LIN {X 0,Y 178.963,Z 581.271,A -85,B 0,C 180,E1 -22404.933,E2 -22404.933} C_VEL
LIN {X 0,Y 179.094,Z 587.177,A -85,B 0,C 180,E1 -22407.754,E2 -22407.754} C_VEL
LIN {X 0,Y 179.064,Z 591.005,A -85,B 0,C 180,E1 -22410.003,E2 -22410.003} C_VEL
LIN {X 0,Y 178.631,Z 594.089,A -85,B 0,C 180,E1 -22412.257,E2 -22412.257} C_VEL
LIN {X 0,Y 177.778,Z 597.609,A -85,B 0,C 180,E1 -22415.674,E2 -22415.674} C_VEL
LIN {X 0,Y 177.413,Z 600.176,A -85,B 0,C 180,E1 -22419.12,E2 -22419.12} C_VEL
LIN {X 0,Y 177.958,Z 602.371,A -85,B 0,C 180,E1 -22423.709,E2 -22423.709} C_VEL
LIN {X 0,Y 180.059,Z 603.293,A -85,B 0,C 180,E1 -22428.198,E2 -22428.198} C_VEL
LIN {X 0,Y 183.553,Z 602.927,A -85,B 0,C 180,E1 -22432.515,E2 -22432.515} C_VEL
LIN {X 0,Y 188.306,Z 601.288,A -85,B 0,C 180,E1 -22436.609,E2 -22436.609} C_VEL
LIN {X 0,Y 194.454,Z 598.389,A -85,B 0,C 180,E1 -22440.4,E2 -22440.4} C_VEL
LIN {X 0,Y 201.914,Z 594.146,A -85,B 0,C 180,E1 -22443.845,E2 -22443.845} C_VEL
LIN {X 0,Y 210.351,Z 588.495,A -85,B 0,C 180,E1 -22446.972,E2 -22446.972} C_VEL
LIN {X 0,Y 217.836,Z 582.763,A -85,B 0,C 180,E1 -22449.257,E2 -22449.257} C_VEL
LIN {X 0,Y 227.369,Z 574.527,A -85,B 0,C 180,E1 -22451.651,E2 -22451.651} C_VEL
LIN {X 0,Y 235.426,Z 566.669,A -85,B 0,C 180,E1 -22453.364,E2 -22453.364} C_VEL
LIN {X 0,Y 244.098,Z 557.229,A -85,B 0,C 180,E1 -22454.864,E2 -22454.864} C_VEL
LIN {X 0,Y 253.168,Z 545.908,A -85,B 0,C 180,E1 -22456.203,E2 -22456.203} C_VEL
LIN {X 0,Y 251.587,Z 547.776,A -85,B 0,C 180,E1 -22456.707,E2 -22456.707} C_VEL
LIN {X 0,Y 243.286,Z 557.033,A -85,B 0,C 180,E1 -22458.362,E2 -22458.362} C_VEL
LIN {X 0,Y 235.512,Z 564.518,A -85,B 0,C 180,E1 -22460.089,E2 -22460.089} C_VEL
LIN {X 0,Y 228.038,Z 570.729,A -85,B 0,C 180,E1 -22461.947,E2 -22461.947} C_VEL
LIN {X 0,Y 220.975,Z 575.798,A -85,B 0,C 180,E1 -22463.957,E2 -22463.957} C_VEL
LIN {X 0,Y 212.204,Z 580.994,A -85,B 0,C 180,E1 -22466.875,E2 -22466.875} C_VEL
LIN {X 0,Y 206.132,Z 583.851,A -85,B 0,C 180,E1 -22469.241,E2 -22469.241} C_VEL
LIN {X 0,Y 198.857,Z 586.335,A -85,B 0,C 180,E1 -22472.648,E2 -22472.648} C_VEL
LIN {X 0,Y 192.485,Z 587.392,A -85,B 0,C 180,E1 -22476.319,E2 -22476.319} C_VEL
LIN {X 0,Y 187.209,Z 586.992,A -85,B 0,C 180,E1 -22480.253,E2 -22480.253} C_VEL
LIN {X 0,Y 182.885,Z 585.199,A -85,B 0,C 180,E1 -22484.395,E2 -22484.395} C_VEL
LIN {X 0,Y 181.145,Z 583.766,A -85,B 0,C 180,E1 -22486.539,E2 -22486.539} C_VEL
LIN {X 0,Y 178.883,Z 579.753,A -85,B 0,C 180,E1 -22490.958,E2 -22490.958} C_VEL
LIN {X 0,Y 177.692,Z 575.71,A -85,B 0,C 180,E1 -22494.325,E2 -22494.325} C_VEL
LIN {X 0,Y 176.868,Z 568.695,A -85,B 0,C 180,E1 -22498.861,E2 -22498.861} C_VEL
LIN {X 0,Y 176.997,Z 560.839,A -85,B 0,C 180,E1 -22502.845,E2 -22502.845} C_VEL
LIN {X 0,Y 177.27,Z 552.453,A -85,B 0,C 180,E1 -22506.249,E2 -22506.249} C_VEL
LIN {X 0,Y 177.78,Z 543.801,A -85,B 0,C 180,E1 -22509.158,E2 -22509.158} C_VEL
LIN {X 0,Y 178.492,Z 533.877,A -85,B 0,C 180,E1 -22511.93,E2 -22511.93} C_VEL
LIN {X 0,Y 179.517,Z 521.445,A -85,B 0,C 180,E1 -22514.742,E2 -22514.742} C_VEL
LIN {X 0,Y 180.559,Z 509.146,A -85,B 0,C 180,E1 -22516.973,E2 -22516.973} C_VEL
LIN {X 0,Y 181.504,Z 495.349,A -85,B 0,C 180,E1 -22518.922,E2 -22518.922} C_VEL
LIN {X 0,Y 182.391,Z 480.871,A -85,B 0,C 180,E1 -22520.438,E2 -22520.438} C_VEL
LIN {X 0,Y 184.893,Z 424.724,A -85,B 0,C 180,E1 -22524.498,E2 -22524.498} C_VEL
LIN {X 0,Y 185.569,Z 410.627,A -85,B 0,C 180,E1 -22525.472,E2 -22525.472} C_VEL
LIN {X 0,Y 178.743,Z 384.831,A -85,B 0,C 180,E1 -22527.528,E2 -22527.528} C_VEL
LIN {X 0,Y 178.643,Z 384.231,A -85,B 0,C 180,E1 -22527.61,E2 -22527.61} C_VEL
LIN {X 0,Y 178.494,Z 384.245,A -85,B 0,C 180,E1 -22533.452,E2 -22533.452} C_VEL
LIN {X 0,Y 178.401,Z 384.26,A -85,B 0,C 180,E1 -22539.073,E2 -22539.073} C_VEL
LIN {X 0,Y 178.404,Z 384.258,A -85,B 0,C 180,E1 -22542.043,E2 -22542.043} C_VEL
LIN {X 0,Y 178.399,Z 384.261,A -85,B 0,C 180,E1 -22545.162,E2 -22545.162} C_VEL
LIN {X 0,Y 178.415,Z 384.259,A -85,B 0,C 180,E1 -22548.455,E2 -22548.455} C_VEL
LIN {X 0,Y 178.468,Z 384.251,A -85,B 0,C 180,E1 -22551.961,E2 -22551.961} C_VEL
LIN {X 0,Y 178.495,Z 384.249,A -85,B 0,C 180,E1 -22556.546,E2 -22556.546} C_VEL
LIN {X 0,Y 178.527,Z 384.242,A -85,B 0,C 180,E1 -22560.004,E2 -22560.004} C_VEL
LIN {X 0,Y 178.538,Z 384.244,A -85,B 0,C 180,E1 -22564.873,E2 -22564.873} C_VEL
LIN {X 0,Y 178.627,Z 384.233,A -85,B 0,C 180,E1 -22570.781,E2 -22570.781} C_VEL
LIN {X 0,Y 178.662,Z 384.225,A -85,B 0,C 180,E1 -22576.346,E2 -22576.346} C_VEL
LIN {X 0,Y 178.914,Z 384.197,A -85,B 0,C 180,E1 -22580.957,E2 -22580.957} C_VEL
LIN {X 0,Y 179.155,Z 384.166,A -85,B 0,C 180,E1 -22587.749,E2 -22587.749} C_VEL
LIN {X 0,Y 179.374,Z 384.143,A -85,B 0,C 180,E1 -22589.997,E2 -22589.997} C_VEL
LIN {X 0,Y 178.878,Z 384.198,A -85,B 0,C 180,E1 -22594.504,E2 -22594.504} C_VEL
LIN {X 0,Y 178.978,Z 384.189,A -85,B 0,C 180,E1 -22599.034,E2 -22599.034} C_VEL
LIN {X 0,Y 178.686,Z 384.222,A -85,B 0,C 180,E1 -22603.647,E2 -22603.647} C_VEL
LIN {X 0,Y 178.648,Z 384.231,A -85,B 0,C 180,E1 -22608.341,E2 -22608.341} C_VEL
LIN {X 0,Y 178.509,Z 384.245,A -85,B 0,C 180,E1 -22613.182,E2 -22613.182} C_VEL
LIN {X 0,Y 178.484,Z 384.25,A -85,B 0,C 180,E1 -22618.194,E2 -22618.194} C_VEL
LIN {X 0,Y 178.475,Z 384.246,A -85,B 0,C 180,E1 -22620.788,E2 -22620.788} C_VEL
LIN {X 0,Y 178.481,Z 384.252,A -85,B 0,C 180,E1 -22624.217,E2 -22624.217} C_VEL
LIN {X 0,Y 178.48,Z 384.248,A -85,B 0,C 180,E1 -22629.049,E2 -22629.049} C_VEL
LIN {X 0,Y 178.509,Z 384.249,A -85,B 0,C 180,E1 -22632.009,E2 -22632.009} C_VEL
LIN {X 0,Y 178.524,Z 384.246,A -85,B 0,C 180,E1 -22635.118,E2 -22635.118} C_VEL
LIN {X 0,Y 178.513,Z 384.243,A -85,B 0,C 180,E1 -22638.415,E2 -22638.415} C_VEL
LIN {X 0,Y 178.481,Z 384.253,A -85,B 0,C 180,E1 -22643.797,E2 -22643.797} C_VEL
LIN {X 0,Y 178.484,Z 384.246,A -85,B 0,C 180,E1 -22646.546,E2 -22646.546} C_VEL
LIN {X 0,Y 178.515,Z 384.248,A -85,B 0,C 180,E1 -22650.005,E2 -22650.005} C_VEL
LIN {X 0,Y 178.527,Z 384.243,A -85,B 0,C 180,E1 -22654.875,E2 -22654.875} C_VEL
LIN {X 0,Y 178.615,Z 384.235,A -85,B 0,C 180,E1 -22660.783,E2 -22660.783} C_VEL
LIN {X 0,Y 178.673,Z 384.226,A -85,B 0,C 180,E1 -22666.349,E2 -22666.349} C_VEL
LIN {X 0,Y 178.97,Z 384.19,A -85,B 0,C 180,E1 -22670.963,E2 -22670.963} C_VEL
LIN {X 0,Y 179.148,Z 384.17,A -85,B 0,C 180,E1 -22677.752,E2 -22677.752} C_VEL
LIN {X 0,Y 179.364,Z 384.14,A -85,B 0,C 180,E1 -22680,E2 -22680} C_VEL
LIN {X 0,Y 178.87,Z 384.201,A -85,B 0,C 180,E1 -22684.507,E2 -22684.507} C_VEL
LIN {X 0,Y 178.97,Z 384.19,A -85,B 0,C 180,E1 -22689.038,E2 -22689.038} C_VEL
LIN {X 0,Y 178.68,Z 384.228,A -85,B 0,C 180,E1 -22693.651,E2 -22693.651} C_VEL
LIN {X 0,Y 178.663,Z 384.226,A -85,B 0,C 180,E1 -22698.343,E2 -22698.343} C_VEL
LIN {X 0,Y 178.506,Z 384.249,A -85,B 0,C 180,E1 -22703.186,E2 -22703.186} C_VEL
LIN {X 0,Y 178.478,Z 384.246,A -85,B 0,C 180,E1 -22708.199,E2 -22708.199} C_VEL
LIN {X 0,Y 178.47,Z 384.251,A -85,B 0,C 180,E1 -22710.793,E2 -22710.793} C_VEL
LIN {X 0,Y 178.478,Z 384.251,A -85,B 0,C 180,E1 -22714.221,E2 -22714.221} C_VEL
LIN {X 0,Y 178.49,Z 384.249,A -85,B 0,C 180,E1 -22719.05,E2 -22719.05} C_VEL
LIN {X 0,Y 178.515,Z 384.247,A -85,B 0,C 180,E1 -22722.012,E2 -22722.012} C_VEL
LIN {X 0,Y 178.525,Z 384.244,A -85,B 0,C 180,E1 -22725.122,E2 -22725.122} C_VEL
LIN {X 0,Y 178.512,Z 384.246,A -85,B 0,C 180,E1 -22728.42,E2 -22728.42} C_VEL
LIN {X 0,Y 178.785,Z 384.32,A -85,B 0,C 180,E1 -22735.035,E2 -22735.035} C_VEL
LIN {X 0,Y 181.805,Z 398.712,A -85,B 0,C 180,E1 -22741.314,E2 -22741.314} C_VEL
LIN {X 0,Y 182.169,Z 424.055,A -85,B 0,C 180,E1 -22743.124,E2 -22743.124} C_VEL
LIN {X 0,Y 184.78,Z 459.469,A -85,B 0,C 180,E1 -22745.699,E2 -22745.699} C_VEL
LIN {X 0,Y 182.685,Z 509.123,A -85,B 0,C 180,E1 -22749.378,E2 -22749.378} C_VEL
LIN {X 0,Y 182.078,Z 520.419,A -85,B 0,C 180,E1 -22750.557,E2 -22750.557} C_VEL
LIN {X 0,Y 181.174,Z 532.641,A -85,B 0,C 180,E1 -22752.216,E2 -22752.216} C_VEL
LIN {X 0,Y 180.286,Z 545.376,A -85,B 0,C 180,E1 -22754.457,E2 -22754.457} C_VEL
LIN {X 0,Y 179.53,Z 556.851,A -85,B 0,C 180,E1 -22756.995,E2 -22756.995} C_VEL
LIN {X 0,Y 179.034,Z 567.273,A -85,B 0,C 180,E1 -22759.861,E2 -22759.861} C_VEL
LIN {X 0,Y 178.932,Z 573.096,A -85,B 0,C 180,E1 -22761.758,E2 -22761.758} C_VEL
LIN {X 0,Y 178.207,Z 576.828,A -85,B 0,C 180,E1 -22763.223,E2 -22763.223} C_VEL
LIN {X 0,Y 175.554,Z 582.018,A -85,B 0,C 180,E1 -22765.819,E2 -22765.819} C_VEL
LIN {X 0,Y 172.593,Z 587.441,A -85,B 0,C 180,E1 -22769.225,E2 -22769.225} C_VEL
LIN {X 0,Y 172.256,Z 589.213,A -85,B 0,C 180,E1 -22770.414,E2 -22770.414} C_VEL
LIN {X 0,Y 171.912,Z 591.86,A -85,B 0,C 180,E1 -22772.346,E2 -22772.346} C_VEL
LIN {X 0,Y 170.974,Z 595.636,A -85,B 0,C 180,E1 -22775.901,E2 -22775.901} C_VEL
LIN {X 0,Y 170.568,Z 598.473,A -85,B 0,C 180,E1 -22779.489,E2 -22779.489} C_VEL
LIN {X 0,Y 171.167,Z 600.987,A -85,B 0,C 180,E1 -22784.265,E2 -22784.265} C_VEL
LIN {X 0,Y 173.363,Z 602.236,A -85,B 0,C 180,E1 -22788.927,E2 -22788.927} C_VEL
LIN {X 0,Y 177.015,Z 602.255,A -85,B 0,C 180,E1 -22793.395,E2 -22793.395} C_VEL
LIN {X 0,Y 181.985,Z 601.049,A -85,B 0,C 180,E1 -22797.611,E2 -22797.611} C_VEL
LIN {X 0,Y 188.369,Z 598.627,A -85,B 0,C 180,E1 -22801.492,E2 -22801.492} C_VEL
LIN {X 0,Y 196.103,Z 594.92,A -85,B 0,C 180,E1 -22804.991,E2 -22804.991} C_VEL
LIN {X 0,Y 204.813,Z 589.857,A -85,B 0,C 180,E1 -22808.148,E2 -22808.148} C_VEL
LIN {X 0,Y 214.431,Z 583.262,A -85,B 0,C 180,E1 -22810.96,E2 -22810.96} C_VEL
LIN {X 0,Y 223.605,Z 576.089,A -85,B 0,C 180,E1 -22813.129,E2 -22813.129} C_VEL
LIN {X 0,Y 231.913,Z 568.759,A -85,B 0,C 180,E1 -22814.798,E2 -22814.798} C_VEL
LIN {X 0,Y 241.255,Z 559.52,A -85,B 0,C 180,E1 -22816.309,E2 -22816.309} C_VEL
LIN {X 0,Y 242.337,Z 558.359,A -85,B 0,C 180,E1 -22816.473,E2 -22816.473} C_VEL
LIN {X 0,Y 241.229,Z 559.378,A -85,B 0,C 180,E1 -22816.85,E2 -22816.85} C_VEL
LIN {X 0,Y 231.935,Z 567.506,A -85,B 0,C 180,E1 -22818.771,E2 -22818.771} C_VEL
LIN {X 0,Y 222.926,Z 574.186,A -85,B 0,C 180,E1 -22820.911,E2 -22820.911} C_VEL
LIN {X 0,Y 213.281,Z 580.016,A -85,B 0,C 180,E1 -22823.62,E2 -22823.62} C_VEL
LIN {X 0,Y 204.438,Z 584.223,A -85,B 0,C 180,E1 -22826.63,E2 -22826.63} C_VEL
LIN {X 0,Y 196.376,Z 586.894,A -85,B 0,C 180,E1 -22829.931,E2 -22829.931} C_VEL
LIN {X 0,Y 189.254,Z 588.163,A -85,B 0,C 180,E1 -22833.537,E2 -22833.537} C_VEL
LIN {X 0,Y 183.156,Z 588.055,A -85,B 0,C 180,E1 -22837.436,E2 -22837.436} C_VEL
LIN {X 0,Y 178.15,Z 586.509,A -85,B 0,C 180,E1 -22841.603,E2 -22841.603} C_VEL
LIN {X 0,Y 174.259,Z 583.552,A -85,B 0,C 180,E1 -22845.996,E2 -22845.996} C_VEL
LIN {X 0,Y 171.903,Z 579.165,A -85,B 0,C 180,E1 -22850.588,E2 -22850.588} C_VEL
LIN {X 0,Y 170.703,Z 574.779,A -85,B 0,C 180,E1 -22854.092,E2 -22854.092} C_VEL
LIN {X 0,Y 169.924,Z 568.358,A -85,B 0,C 180,E1 -22858.222,E2 -22858.222} C_VEL
LIN {X 0,Y 169.983,Z 560.308,A -85,B 0,C 180,E1 -22862.369,E2 -22862.369} C_VEL
LIN {X 0,Y 170.252,Z 551.734,A -85,B 0,C 180,E1 -22865.923,E2 -22865.923} C_VEL
LIN {X 0,Y 170.847,Z 541.719,A -85,B 0,C 180,E1 -22869.302,E2 -22869.302} C_VEL
LIN {X 0,Y 171.676,Z 530.406,A -85,B 0,C 180,E1 -22872.411,E2 -22872.411} C_VEL
LIN {X 0,Y 172.687,Z 518.564,A -85,B 0,C 180,E1 -22875.037,E2 -22875.037} C_VEL
LIN {X 0,Y 173.737,Z 505.427,A -85,B 0,C 180,E1 -22877.357,E2 -22877.357} C_VEL
LIN {X 0,Y 174.736,Z 490.405,A -85,B 0,C 180,E1 -22879.379,E2 -22879.379} C_VEL
LIN {X 0,Y 175.616,Z 474.732,A -85,B 0,C 180,E1 -22880.88,E2 -22880.88} C_VEL
LIN {X 0,Y 178.467,Z 411.765,A -85,B 0,C 180,E1 -22885.566,E2 -22885.566} C_VEL
LIN {X 0,Y 171.642,Z 385.486,A -85,B 0,C 180,E1 -22887.731,E2 -22887.731} C_VEL
LIN {X 0,Y 171.599,Z 385.109,A -85,B 0,C 180,E1 -22887.786,E2 -22887.786} C_VEL
LIN {X 0,Y 171.424,Z 385.128,A -85,B 0,C 180,E1 -22892.206,E2 -22892.206} C_VEL
LIN {X 0,Y 171.399,Z 385.132,A -85,B 0,C 180,E1 -22895.033,E2 -22895.033} C_VEL
LIN {X 0,Y 171.363,Z 385.137,A -85,B 0,C 180,E1 -22898.806,E2 -22898.806} C_VEL
LIN {X 0,Y 171.326,Z 385.143,A -85,B 0,C 180,E1 -22904.215,E2 -22904.215} C_VEL
LIN {X 0,Y 171.349,Z 385.137,A -85,B 0,C 180,E1 -22908.982,E2 -22908.982} C_VEL
LIN {X 0,Y 171.418,Z 385.129,A -85,B 0,C 180,E1 -22912.046,E2 -22912.046} C_VEL
LIN {X 0,Y 171.415,Z 385.131,A -85,B 0,C 180,E1 -22915.084,E2 -22915.084} C_VEL
LIN {X 0,Y 171.454,Z 385.126,A -85,B 0,C 180,E1 -22920.532,E2 -22920.532} C_VEL
LIN {X 0,Y 171.462,Z 385.126,A -85,B 0,C 180,E1 -22925.799,E2 -22925.799} C_VEL
LIN {X 0,Y 171.583,Z 385.11,A -85,B 0,C 180,E1 -22930.869,E2 -22930.869} C_VEL
LIN {X 0,Y 171.58,Z 385.11,A -85,B 0,C 180,E1 -22935.77,E2 -22935.77} C_VEL
LIN {X 0,Y 171.85,Z 385.078,A -85,B 0,C 180,E1 -22940.582,E2 -22940.582} C_VEL
LIN {X 0,Y 171.819,Z 385.077,A -85,B 0,C 180,E1 -22945.305,E2 -22945.305} C_VEL
LIN {X 0,Y 172.336,Z 385.02,A -85,B 0,C 180,E1 -22949.997,E2 -22949.997} C_VEL
LIN {X 0,Y 171.827,Z 385.076,A -85,B 0,C 180,E1 -22954.689,E2 -22954.689} C_VEL
LIN {X 0,Y 171.91,Z 385.07,A -85,B 0,C 180,E1 -22959.409,E2 -22959.409} C_VEL
LIN {X 0,Y 171.609,Z 385.106,A -85,B 0,C 180,E1 -22964.222,E2 -22964.222} C_VEL
LIN {X 0,Y 171.543,Z 385.116,A -85,B 0,C 180,E1 -22969.56,E2 -22969.56} C_VEL
LIN {X 0,Y 171.466,Z 385.126,A -85,B 0,C 180,E1 -22975.614,E2 -22975.614} C_VEL
LIN {X 0,Y 171.438,Z 385.123,A -85,B 0,C 180,E1 -22980.584,E2 -22980.584} C_VEL
LIN {X 0,Y 171.435,Z 385.129,A -85,B 0,C 180,E1 -22985.021,E2 -22985.021} C_VEL
LIN {X 0,Y 171.433,Z 385.125,A -85,B 0,C 180,E1 -22988.839,E2 -22988.839} C_VEL
LIN {X 0,Y 171.447,Z 385.128,A -85,B 0,C 180,E1 -22994.172,E2 -22994.172} C_VEL
LIN {X 0,Y 171.429,Z 385.125,A -85,B 0,C 180,E1 -22999.009,E2 -22999.009} C_VEL
LIN {X 0,Y 171.437,Z 385.13,A -85,B 0,C 180,E1 -23002.054,E2 -23002.054} C_VEL
LIN {X 0,Y 171.434,Z 385.128,A -85,B 0,C 180,E1 -23005.07,E2 -23005.07} C_VEL
LIN {X 0,Y 171.442,Z 385.128,A -85,B 0,C 180,E1 -23010.533,E2 -23010.533} C_VEL
LIN {X 0,Y 171.45,Z 385.124,A -85,B 0,C 180,E1 -23015.801,E2 -23015.801} C_VEL
LIN {X 0,Y 171.571,Z 385.112,A -85,B 0,C 180,E1 -23020.871,E2 -23020.871} C_VEL
LIN {X 0,Y 171.586,Z 385.109,A -85,B 0,C 180,E1 -23025.774,E2 -23025.774} C_VEL
LIN {X 0,Y 171.902,Z 385.07,A -85,B 0,C 180,E1 -23030.588,E2 -23030.588} C_VEL
LIN {X 0,Y 171.82,Z 385.08,A -85,B 0,C 180,E1 -23035.308,E2 -23035.308} C_VEL
LIN {X 0,Y 172.327,Z 385.016,A -85,B 0,C 180,E1 -23040,E2 -23040} C_VEL
LIN {X 0,Y 171.82,Z 385.08,A -85,B 0,C 180,E1 -23044.693,E2 -23044.693} C_VEL
LIN {X 0,Y 171.902,Z 385.07,A -85,B 0,C 180,E1 -23049.412,E2 -23049.412} C_VEL
LIN {X 0,Y 171.605,Z 385.108,A -85,B 0,C 180,E1 -23054.225,E2 -23054.225} C_VEL
LIN {X 0,Y 171.55,Z 385.111,A -85,B 0,C 180,E1 -23059.576,E2 -23059.576} C_VEL
LIN {X 0,Y 171.461,Z 385.126,A -85,B 0,C 180,E1 -23065.618,E2 -23065.618} C_VEL
LIN {X 0,Y 171.433,Z 385.127,A -85,B 0,C 180,E1 -23070.587,E2 -23070.587} C_VEL
LIN {X 0,Y 171.402,Z 385.134,A -85,B 0,C 180,E1 -23075.033,E2 -23075.033} C_VEL
LIN {X 0,Y 171.441,Z 385.126,A -85,B 0,C 180,E1 -23078.847,E2 -23078.847} C_VEL
LIN {X 0,Y 171.45,Z 385.125,A -85,B 0,C 180,E1 -23084.176,E2 -23084.176} C_VEL
LIN {X 0,Y 171.433,Z 385.13,A -85,B 0,C 180,E1 -23089.014,E2 -23089.014} C_VEL
LIN {X 0,Y 171.759,Z 385.193,A -85,B 0,C 180,E1 -23095.141,E2 -23095.141} C_VEL
LIN {X 0,Y 174.463,Z 397.947,A -85,B 0,C 180,E1 -23101.01,E2 -23101.01} C_VEL
LIN {X 0,Y 174.826,Z 402.006,A -85,B 0,C 180,E1 -23101.324,E2 -23101.324} C_VEL
LIN {X 0,Y 174.995,Z 422.325,A -85,B 0,C 180,E1 -23102.846,E2 -23102.846} C_VEL
LIN {X 0,Y 177.645,Z 459.917,A -85,B 0,C 180,E1 -23105.708,E2 -23105.708} C_VEL
LIN {X 0,Y 175.628,Z 508.529,A -85,B 0,C 180,E1 -23109.507,E2 -23109.507} C_VEL
LIN {X 0,Y 175,Z 520.309,A -85,B 0,C 180,E1 -23110.806,E2 -23110.806} C_VEL
LIN {X 0,Y 174.046,Z 533.204,A -85,B 0,C 180,E1 -23112.677,E2 -23112.677} C_VEL
LIN {X 0,Y 173.248,Z 545.71,A -85,B 0,C 180,E1 -23115.015,E2 -23115.015} C_VEL
LIN {X 0,Y 172.539,Z 556.89,A -85,B 0,C 180,E1 -23117.656,E2 -23117.656} C_VEL
LIN {X 0,Y 172.158,Z 567.042,A -85,B 0,C 180,E1 -23120.605,E2 -23120.605} C_VEL
LIN {X 0,Y 172.027,Z 575.333,A -85,B 0,C 180,E1 -23123.552,E2 -23123.552} C_VEL
LIN {X 0,Y 172.268,Z 582.181,A -85,B 0,C 180,E1 -23126.494,E2 -23126.494} C_VEL
LIN {X 0,Y 172.329,Z 586.641,A -85,B 0,C 180,E1 -23128.834,E2 -23128.834} C_VEL
LIN {X 0,Y 172.256,Z 589.213,A -85,B 0,C 180,E1 -23130.414,E2 -23130.414} C_VEL
LIN {X 0,Y 171.81,Z 590.823,A -85,B 0,C 180,E1 -23131.598,E2 -23131.598} C_VEL
LIN {X 0,Y 170.804,Z 592.098,A -85,B 0,C 180,E1 -23132.793,E2 -23132.793} C_VEL
LIN {X 0,Y 167.929,Z 594.009,A -85,B 0,C 180,E1 -23135.219,E2 -23135.219} C_VEL
LIN {X 0,Y 165.072,Z 595.457,A -85,B 0,C 180,E1 -23137.782,E2 -23137.782} C_VEL
LIN {X 0,Y 163.869,Z 596.57,A -85,B 0,C 180,E1 -23139.805,E2 -23139.805} C_VEL
LIN {X 0,Y 163.779,Z 596.978,A -85,B 0,C 180,E1 -23140.492,E2 -23140.492} C_VEL
LIN {X 0,Y 164.423,Z 599.434,A -85,B 0,C 180,E1 -23144.863,E2 -23144.863} C_VEL
LIN {X 0,Y 166.719,Z 601.046,A -85,B 0,C 180,E1 -23149.712,E2 -23149.712} C_VEL
LIN {X 0,Y 170.527,Z 601.456,A -85,B 0,C 180,E1 -23154.342,E2 -23154.342} C_VEL
LIN {X 0,Y 175.747,Z 600.682,A -85,B 0,C 180,E1 -23158.68,E2 -23158.68} C_VEL
LIN {X 0,Y 182.364,Z 598.728,A -85,B 0,C 180,E1 -23162.655,E2 -23162.655} C_VEL
LIN {X 0,Y 190.362,Z 595.548,A -85,B 0,C 180,E1 -23166.21,E2 -23166.21} C_VEL
LIN {X 0,Y 199.335,Z 591.051,A -85,B 0,C 180,E1 -23169.395,E2 -23169.395} C_VEL
LIN {X 0,Y 209.219,Z 585.134,A -85,B 0,C 180,E1 -23172.211,E2 -23172.211} C_VEL
LIN {X 0,Y 218.617,Z 578.65,A -85,B 0,C 180,E1 -23174.366,E2 -23174.366} C_VEL
LIN {X 0,Y 227.078,Z 572.026,A -85,B 0,C 180,E1 -23176.022,E2 -23176.022} C_VEL
LIN {X 0,Y 231.547,Z 568.232,A -85,B 0,C 180,E1 -23176.76,E2 -23176.76} C_VEL
LIN {X 0,Y 223.107,Z 574.203,A -85,B 0,C 180,E1 -23178.584,E2 -23178.584} C_VEL
LIN {X 0,Y 215.287,Z 578.909,A -85,B 0,C 180,E1 -23180.463,E2 -23180.463} C_VEL
LIN {X 0,Y 207.915,Z 582.624,A -85,B 0,C 180,E1 -23182.523,E2 -23182.523} C_VEL
LIN {X 0,Y 198.755,Z 586.235,A -85,B 0,C 180,E1 -23185.544,E2 -23185.544} C_VEL
LIN {X 0,Y 190.391,Z 588.402,A -85,B 0,C 180,E1 -23188.883,E2 -23188.883} C_VEL
LIN {X 0,Y 182.994,Z 589.156,A -85,B 0,C 180,E1 -23192.557,E2 -23192.557} C_VEL
LIN {X 0,Y 176.649,Z 588.558,A -85,B 0,C 180,E1 -23196.556,E2 -23196.556} C_VEL
LIN {X 0,Y 171.44,Z 586.601,A -85,B 0,C 180,E1 -23200.855,E2 -23200.855} C_VEL
LIN {X 0,Y 167.391,Z 583.202,A -85,B 0,C 180,E1 -23205.409,E2 -23205.409} C_VEL
LIN {X 0,Y 164.947,Z 578.371,A -85,B 0,C 180,E1 -23210.187,E2 -23210.187} C_VEL
LIN {X 0,Y 163.716,Z 573.659,A -85,B 0,C 180,E1 -23213.839,E2 -23213.839} C_VEL
LIN {X 0,Y 162.966,Z 566.838,A -85,B 0,C 180,E1 -23218.146,E2 -23218.146} C_VEL
LIN {X 0,Y 163.065,Z 558.318,A -85,B 0,C 180,E1 -23222.47,E2 -23222.47} C_VEL
LIN {X 0,Y 163.369,Z 549.245,A -85,B 0,C 180,E1 -23226.174,E2 -23226.174} C_VEL
LIN {X 0,Y 163.982,Z 539.246,A -85,B 0,C 180,E1 -23229.511,E2 -23229.511} C_VEL
LIN {X 0,Y 164.804,Z 527.785,A -85,B 0,C 180,E1 -23232.624,E2 -23232.624} C_VEL
LIN {X 0,Y 165.853,Z 515.28,A -85,B 0,C 180,E1 -23235.357,E2 -23235.357} C_VEL
LIN {X 0,Y 166.792,Z 503.141,A -85,B 0,C 180,E1 -23237.471,E2 -23237.471} C_VEL
LIN {X 0,Y 167.681,Z 489.929,A -85,B 0,C 180,E1 -23239.272,E2 -23239.272} C_VEL
LIN {X 0,Y 168.527,Z 474.924,A -85,B 0,C 180,E1 -23240.761,E2 -23240.761} C_VEL
LIN {X 0,Y 171.372,Z 412.584,A -85,B 0,C 180,E1 -23245.662,E2 -23245.662} C_VEL
LIN {X 0,Y 164.916,Z 387.845,A -85,B 0,C 180,E1 -23247.768,E2 -23247.768} C_VEL
LIN {X 0,Y 164.536,Z 385.989,A -85,B 0,C 180,E1 -23247.975,E2 -23247.975} C_VEL
LIN {X 0,Y 164.333,Z 386.009,A -85,B 0,C 180,E1 -23253.777,E2 -23253.777} C_VEL
LIN {X 0,Y 164.3,Z 386.019,A -85,B 0,C 180,E1 -23256.788,E2 -23256.788} C_VEL
LIN {X 0,Y 164.296,Z 386.018,A -85,B 0,C 180,E1 -23259.914,E2 -23259.914} C_VEL
LIN {X 0,Y 164.285,Z 386.017,A -85,B 0,C 180,E1 -23263.34,E2 -23263.34} C_VEL
LIN {X 0,Y 164.297,Z 386.018,A -85,B 0,C 180,E1 -23266.807,E2 -23266.807} C_VEL
LIN {X 0,Y 164.31,Z 386.013,A -85,B 0,C 180,E1 -23270.346,E2 -23270.346} C_VEL
LIN {X 0,Y 164.348,Z 386.014,A -85,B 0,C 180,E1 -23274.34,E2 -23274.34} C_VEL
LIN {X 0,Y 164.395,Z 386,A -85,B 0,C 180,E1 -23279.133,E2 -23279.133} C_VEL
LIN {X 0,Y 164.42,Z 386.003,A -85,B 0,C 180,E1 -23284.692,E2 -23284.692} C_VEL
LIN {X 0,Y 164.488,Z 385.994,A -85,B 0,C 180,E1 -23290.048,E2 -23290.048} C_VEL
LIN {X 0,Y 164.527,Z 385.987,A -85,B 0,C 180,E1 -23295.147,E2 -23295.147} C_VEL
LIN {X 0,Y 164.771,Z 385.962,A -85,B 0,C 180,E1 -23300.174,E2 -23300.174} C_VEL
LIN {X 0,Y 164.834,Z 385.951,A -85,B 0,C 180,E1 -23302.648,E2 -23302.648} C_VEL
LIN {X 0,Y 165.05,Z 385.922,A -85,B 0,C 180,E1 -23307.557,E2 -23307.557} C_VEL
LIN {X 0,Y 165.299,Z 385.896,A -85,B 0,C 180,E1 -23309.997,E2 -23309.997} C_VEL
LIN {X 0,Y 164.778,Z 385.954,A -85,B 0,C 180,E1 -23314.891,E2 -23314.891} C_VEL
LIN {X 0,Y 164.863,Z 385.947,A -85,B 0,C 180,E1 -23317.345,E2 -23317.345} C_VEL
LIN {X 0,Y 164.779,Z 385.957,A -85,B 0,C 180,E1 -23321.195,E2 -23321.195} C_VEL
LIN {X 0,Y 164.504,Z 385.993,A -85,B 0,C 180,E1 -23327.398,E2 -23327.398} C_VEL
LIN {X 0,Y 164.471,Z 385.995,A -85,B 0,C 180,E1 -23329.986,E2 -23329.986} C_VEL
LIN {X 0,Y 164.39,Z 386.008,A -85,B 0,C 180,E1 -23336.131,E2 -23336.131} C_VEL
LIN {X 0,Y 164.372,Z 386.003,A -85,B 0,C 180,E1 -23341.226,E2 -23341.226} C_VEL
LIN {X 0,Y 164.357,Z 386.01,A -85,B 0,C 180,E1 -23346.769,E2 -23346.769} C_VEL
LIN {X 0,Y 164.37,Z 386.006,A -85,B 0,C 180,E1 -23349.889,E2 -23349.889} C_VEL
LIN {X 0,Y 164.385,Z 386.008,A -85,B 0,C 180,E1 -23353.381,E2 -23353.381} C_VEL
LIN {X 0,Y 164.391,Z 386.004,A -85,B 0,C 180,E1 -23356.841,E2 -23356.841} C_VEL
LIN {X 0,Y 164.371,Z 386.008,A -85,B 0,C 180,E1 -23360.315,E2 -23360.315} C_VEL
LIN {X 0,Y 164.363,Z 386.009,A -85,B 0,C 180,E1 -23364.328,E2 -23364.328} C_VEL
LIN {X 0,Y 164.384,Z 386.006,A -85,B 0,C 180,E1 -23369.133,E2 -23369.133} C_VEL
LIN {X 0,Y 164.409,Z 386.001,A -85,B 0,C 180,E1 -23374.693,E2 -23374.693} C_VEL
LIN {X 0,Y 164.477,Z 385.997,A -85,B 0,C 180,E1 -23380.05,E2 -23380.05} C_VEL
LIN {X 0,Y 164.528,Z 385.984,A -85,B 0,C 180,E1 -23385.15,E2 -23385.15} C_VEL
LIN {X 0,Y 164.844,Z 385.95,A -85,B 0,C 180,E1 -23390.181,E2 -23390.181} C_VEL
LIN {X 0,Y 164.77,Z 385.957,A -85,B 0,C 180,E1 -23395.107,E2 -23395.107} C_VEL
LIN {X 0,Y 165.289,Z 385.893,A -85,B 0,C 180,E1 -23400,E2 -23400} C_VEL
LIN {X 0,Y 164.77,Z 385.958,A -85,B 0,C 180,E1 -23404.894,E2 -23404.894} C_VEL
LIN {X 0,Y 164.845,Z 385.946,A -85,B 0,C 180,E1 -23409.819,E2 -23409.819} C_VEL
LIN {X 0,Y 164.551,Z 385.987,A -85,B 0,C 180,E1 -23414.849,E2 -23414.849} C_VEL
LIN {X 0,Y 164.468,Z 385.993,A -85,B 0,C 180,E1 -23419.99,E2 -23419.99} C_VEL
LIN {X 0,Y 164.386,Z 386.006,A -85,B 0,C 180,E1 -23426.135,E2 -23426.135} C_VEL
LIN {X 0,Y 164.367,Z 386.01,A -85,B 0,C 180,E1 -23431.229,E2 -23431.229} C_VEL
LIN {X 0,Y 164.347,Z 386.009,A -85,B 0,C 180,E1 -23436.776,E2 -23436.776} C_VEL
LIN {X 0,Y 164.374,Z 386.008,A -85,B 0,C 180,E1 -23439.893,E2 -23439.893} C_VEL
LIN {X 0,Y 164.389,Z 386.007,A -85,B 0,C 180,E1 -23443.387,E2 -23443.387} C_VEL
LIN {X 0,Y 164.391,Z 386.002,A -85,B 0,C 180,E1 -23446.845,E2 -23446.845} C_VEL
LIN {X 0,Y 164.507,Z 385.99,A -85,B 0,C 180,E1 -23453.27,E2 -23453.27} C_VEL
LIN {X 0,Y 164.727,Z 386.154,A -85,B 0,C 180,E1 -23455.333,E2 -23455.333} C_VEL
LIN {X 0,Y 167.177,Z 397.333,A -85,B 0,C 180,E1 -23460.71,E2 -23460.71} C_VEL
LIN {X 0,Y 167.774,Z 401.528,A -85,B 0,C 180,E1 -23461.086,E2 -23461.086} C_VEL
LIN {X 0,Y 167.918,Z 421.862,A -85,B 0,C 180,E1 -23462.684,E2 -23462.684} C_VEL
LIN {X 0,Y 170.571,Z 459.332,A -85,B 0,C 180,E1 -23465.671,E2 -23465.671} C_VEL
LIN {X 0,Y 168.604,Z 507.692,A -85,B 0,C 180,E1 -23469.651,E2 -23469.651} C_VEL
LIN {X 0,Y 168.042,Z 518.867,A -85,B 0,C 180,E1 -23470.932,E2 -23470.932} C_VEL
LIN {X 0,Y 167.102,Z 531.875,A -85,B 0,C 180,E1 -23472.881,E2 -23472.881} C_VEL
LIN {X 0,Y 166.324,Z 544.442,A -85,B 0,C 180,E1 -23475.317,E2 -23475.317} C_VEL
LIN {X 0,Y 165.658,Z 555.605,A -85,B 0,C 180,E1 -23478.038,E2 -23478.038} C_VEL
LIN {X 0,Y 165.356,Z 564.952,A -85,B 0,C 180,E1 -23480.832,E2 -23480.832} C_VEL
LIN {X 0,Y 165.268,Z 573.431,A -85,B 0,C 180,E1 -23483.9,E2 -23483.9} C_VEL
LIN {X 0,Y 165.548,Z 580.431,A -85,B 0,C 180,E1 -23486.961,E2 -23486.961} C_VEL
LIN {X 0,Y 165.575,Z 585.994,A -85,B 0,C 180,E1 -23490.003,E2 -23490.003} C_VEL
LIN {X 0,Y 165.513,Z 587.901,A -85,B 0,C 180,E1 -23491.219,E2 -23491.219} C_VEL
LIN {X 0,Y 164.52,Z 592.33,A -85,B 0,C 180,E1 -23494.904,E2 -23494.904} C_VEL
LIN {X 0,Y 163.783,Z 596.597,A -85,B 0,C 180,E1 -23499.886,E2 -23499.886} C_VEL
LIN {X 0,Y 163.779,Z 596.978,A -85,B 0,C 180,E1 -23500.492,E2 -23500.492} C_VEL
LIN {X 0,Y 163.281,Z 598.066,A -85,B 0,C 180,E1 -23502.524,E2 -23502.524} C_VEL
LIN {X 0,Y 161.316,Z 599.003,A -85,B 0,C 180,E1 -23505.94,E2 -23505.94} C_VEL
LIN {X 0,Y 160.126,Z 599.562,A -85,B 0,C 180,E1 -23509.439,E2 -23509.439} C_VEL
LIN {X 0,Y 160.83,Z 599.943,A -85,B 0,C 180,E1 -23511.524,E2 -23511.524} C_VEL
LIN {X 0,Y 164.106,Z 600.519,A -85,B 0,C 180,E1 -23515.36,E2 -23515.36} C_VEL
LIN {X 0,Y 169.572,Z 600.172,A -85,B 0,C 180,E1 -23519.827,E2 -23519.827} C_VEL
LIN {X 0,Y 176.447,Z 598.677,A -85,B 0,C 180,E1 -23523.895,E2 -23523.895} C_VEL
LIN {X 0,Y 184.692,Z 596.003,A -85,B 0,C 180,E1 -23527.508,E2 -23527.508} C_VEL
LIN {X 0,Y 193.934,Z 592.068,A -85,B 0,C 180,E1 -23530.718,E2 -23530.718} C_VEL
LIN {X 0,Y 204.091,Z 586.807,A -85,B 0,C 180,E1 -23533.531,E2 -23533.531} C_VEL
LIN {X 0,Y 215.12,Z 580.058,A -85,B 0,C 180,E1 -23535.953,E2 -23535.953} C_VEL
LIN {X 0,Y 219.422,Z 577.109,A -85,B 0,C 180,E1 -23536.792,E2 -23536.792} C_VEL
LIN {X 0,Y 218.221,Z 577.672,A -85,B 0,C 180,E1 -23537.443,E2 -23537.443} C_VEL
LIN {X 0,Y 210.192,Z 581.834,A -85,B 0,C 180,E1 -23539.307,E2 -23539.307} C_VEL
LIN {X 0,Y 202.59,Z 585.076,A -85,B 0,C 180,E1 -23541.359,E2 -23541.359} C_VEL
LIN {X 0,Y 193.119,Z 588.095,A -85,B 0,C 180,E1 -23544.389,E2 -23544.389} C_VEL
LIN {X 0,Y 184.449,Z 589.747,A -85,B 0,C 180,E1 -23547.762,E2 -23547.762} C_VEL
LIN {X 0,Y 176.766,Z 590.004,A -85,B 0,C 180,E1 -23551.503,E2 -23551.503} C_VEL
LIN {X 0,Y 170.17,Z 588.916,A -85,B 0,C 180,E1 -23555.606,E2 -23555.606} C_VEL
LIN {X 0,Y 164.765,Z 586.494,A -85,B 0,C 180,E1 -23560.047,E2 -23560.047} C_VEL
LIN {X 0,Y 160.563,Z 582.696,A -85,B 0,C 180,E1 -23564.774,E2 -23564.774} C_VEL
LIN {X 0,Y 158.043,Z 577.414,A -85,B 0,C 180,E1 -23569.754,E2 -23569.754} C_VEL
LIN {X 0,Y 156.771,Z 572.375,A -85,B 0,C 180,E1 -23573.565,E2 -23573.565} C_VEL
LIN {X 0,Y 156.043,Z 565.105,A -85,B 0,C 180,E1 -23578.064,E2 -23578.064} C_VEL
LIN {X 0,Y 156.125,Z 557.517,A -85,B 0,C 180,E1 -23581.934,E2 -23581.934} C_VEL
LIN {X 0,Y 156.321,Z 549.9,A -85,B 0,C 180,E1 -23585.159,E2 -23585.159} C_VEL
LIN {X 0,Y 156.913,Z 539.472,A -85,B 0,C 180,E1 -23588.814,E2 -23588.814} C_VEL
LIN {X 0,Y 157.666,Z 529.086,A -85,B 0,C 180,E1 -23591.799,E2 -23591.799} C_VEL
LIN {X 0,Y 158.682,Z 516.404,A -85,B 0,C 180,E1 -23594.754,E2 -23594.754} C_VEL
LIN {X 0,Y 159.738,Z 502.625,A -85,B 0,C 180,E1 -23597.276,E2 -23597.276} C_VEL
LIN {X 0,Y 160.642,Z 489.136,A -85,B 0,C 180,E1 -23599.154,E2 -23599.154} C_VEL
LIN {X 0,Y 161.491,Z 473.783,A -85,B 0,C 180,E1 -23600.707,E2 -23600.707} C_VEL
LIN {X 0,Y 164.124,Z 412.968,A -85,B 0,C 180,E1 -23605.76,E2 -23605.76} C_VEL
LIN {X 0,Y 158.054,Z 389.582,A -85,B 0,C 180,E1 -23607.834,E2 -23607.834} C_VEL
LIN {X 0,Y 157.493,Z 386.867,A -85,B 0,C 180,E1 -23608.118,E2 -23608.118} C_VEL
LIN {X 0,Y 157.282,Z 386.888,A -85,B 0,C 180,E1 -23612.426,E2 -23612.426} C_VEL
LIN {X 0,Y 157.274,Z 386.895,A -85,B 0,C 180,E1 -23616.448,E2 -23616.448} C_VEL
LIN {X 0,Y 157.198,Z 386.898,A -85,B 0,C 180,E1 -23622.115,E2 -23622.115} C_VEL
LIN {X 0,Y 157.218,Z 386.901,A -85,B 0,C 180,E1 -23627.888,E2 -23627.888} C_VEL
LIN {X 0,Y 157.287,Z 386.891,A -85,B 0,C 180,E1 -23633.541,E2 -23633.541} C_VEL
LIN {X 0,Y 157.299,Z 386.887,A -85,B 0,C 180,E1 -23638.092,E2 -23638.092} C_VEL
LIN {X 0,Y 157.326,Z 386.887,A -85,B 0,C 180,E1 -23643.464,E2 -23643.464} C_VEL
LIN {X 0,Y 157.397,Z 386.875,A -85,B 0,C 180,E1 -23649.665,E2 -23649.665} C_VEL
LIN {X 0,Y 157.457,Z 386.869,A -85,B 0,C 180,E1 -23654.463,E2 -23654.463} C_VEL
LIN {X 0,Y 157.692,Z 386.841,A -85,B 0,C 180,E1 -23659.728,E2 -23659.728} C_VEL
LIN {X 0,Y 157.77,Z 386.832,A -85,B 0,C 180,E1 -23662.317,E2 -23662.317} C_VEL
LIN {X 0,Y 158.261,Z 386.773,A -85,B 0,C 180,E1 -23669.997,E2 -23669.997} C_VEL
LIN {X 0,Y 157.825,Z 386.825,A -85,B 0,C 180,E1 -23677.674,E2 -23677.674} C_VEL
LIN {X 0,Y 157.705,Z 386.838,A -85,B 0,C 180,E1 -23681.359,E2 -23681.359} C_VEL
LIN {X 0,Y 157.477,Z 386.867,A -85,B 0,C 180,E1 -23685.529,E2 -23685.529} C_VEL
LIN {X 0,Y 157.368,Z 386.878,A -85,B 0,C 180,E1 -23690.93,E2 -23690.93} C_VEL
LIN {X 0,Y 157.312,Z 386.888,A -85,B 0,C 180,E1 -23696.682,E2 -23696.682} C_VEL
LIN {X 0,Y 157.28,Z 386.891,A -85,B 0,C 180,E1 -23702.423,E2 -23702.423} C_VEL
LIN {X 0,Y 157.335,Z 386.885,A -85,B 0,C 180,E1 -23706.482,E2 -23706.482} C_VEL
LIN {X 0,Y 157.29,Z 386.892,A -85,B 0,C 180,E1 -23712.08,E2 -23712.08} C_VEL
LIN {X 0,Y 157.308,Z 386.89,A -85,B 0,C 180,E1 -23715.624,E2 -23715.624} C_VEL
LIN {X 0,Y 157.288,Z 386.891,A -85,B 0,C 180,E1 -23721.278,E2 -23721.278} C_VEL
LIN {X 0,Y 157.308,Z 386.888,A -85,B 0,C 180,E1 -23724.494,E2 -23724.494} C_VEL
LIN {X 0,Y 157.29,Z 386.889,A -85,B 0,C 180,E1 -23728.092,E2 -23728.092} C_VEL
LIN {X 0,Y 157.315,Z 386.889,A -85,B 0,C 180,E1 -23733.465,E2 -23733.465} C_VEL
LIN {X 0,Y 157.386,Z 386.882,A -85,B 0,C 180,E1 -23739.666,E2 -23739.666} C_VEL
LIN {X 0,Y 157.454,Z 386.864,A -85,B 0,C 180,E1 -23744.466,E2 -23744.466} C_VEL
LIN {X 0,Y 157.764,Z 386.833,A -85,B 0,C 180,E1 -23749.736,E2 -23749.736} C_VEL
LIN {X 0,Y 157.816,Z 386.822,A -85,B 0,C 180,E1 -23752.323,E2 -23752.323} C_VEL
LIN {X 0,Y 158.251,Z 386.77,A -85,B 0,C 180,E1 -23760,E2 -23760} C_VEL
LIN {X 0,Y 157.817,Z 386.826,A -85,B 0,C 180,E1 -23767.678,E2 -23767.678} C_VEL
LIN {X 0,Y 157.698,Z 386.836,A -85,B 0,C 180,E1 -23771.363,E2 -23771.363} C_VEL
LIN {X 0,Y 157.478,Z 386.87,A -85,B 0,C 180,E1 -23775.532,E2 -23775.532} C_VEL
LIN {X 0,Y 157.364,Z 386.878,A -85,B 0,C 180,E1 -23780.934,E2 -23780.934} C_VEL
LIN {X 0,Y 157.307,Z 386.888,A -85,B 0,C 180,E1 -23786.686,E2 -23786.686} C_VEL
LIN {X 0,Y 157.271,Z 386.893,A -85,B 0,C 180,E1 -23792.429,E2 -23792.429} C_VEL
LIN {X 0,Y 157.321,Z 386.884,A -85,B 0,C 180,E1 -23796.481,E2 -23796.481} C_VEL
LIN {X 0,Y 157.294,Z 386.891,A -85,B 0,C 180,E1 -23802.084,E2 -23802.084} C_VEL
LIN {X 0,Y 157.309,Z 386.884,A -85,B 0,C 180,E1 -23805.629,E2 -23805.629} C_VEL
LIN {X 0,Y 157.356,Z 386.884,A -85,B 0,C 180,E1 -23811.301,E2 -23811.301} C_VEL
LIN {X 0,Y 157.696,Z 386.942,A -85,B 0,C 180,E1 -23815.5,E2 -23815.5} C_VEL
LIN {X 0,Y 159.899,Z 396.817,A -85,B 0,C 180,E1 -23820.456,E2 -23820.456} C_VEL
LIN {X 0,Y 160.665,Z 402.185,A -85,B 0,C 180,E1 -23820.951,E2 -23820.951} C_VEL
LIN {X 0,Y 160.933,Z 424.858,A -85,B 0,C 180,E1 -23822.832,E2 -23822.832} C_VEL
LIN {X 0,Y 163.447,Z 459.569,A -85,B 0,C 180,E1 -23825.732,E2 -23825.732} C_VEL
LIN {X 0,Y 161.516,Z 508.008,A -85,B 0,C 180,E1 -23829.964,E2 -23829.964} C_VEL
LIN {X 0,Y 160.922,Z 519.438,A -85,B 0,C 180,E1 -23831.379,E2 -23831.379} C_VEL
LIN {X 0,Y 160.058,Z 532.078,A -85,B 0,C 180,E1 -23833.42,E2 -23833.42} C_VEL
LIN {X 0,Y 159.374,Z 544.433,A -85,B 0,C 180,E1 -23835.966,E2 -23835.966} C_VEL
LIN {X 0,Y 158.746,Z 555.4,A -85,B 0,C 180,E1 -23838.805,E2 -23838.805} C_VEL
LIN {X 0,Y 158.538,Z 564.607,A -85,B 0,C 180,E1 -23841.719,E2 -23841.719} C_VEL
LIN {X 0,Y 158.593,Z 572.979,A -85,B 0,C 180,E1 -23844.918,E2 -23844.918} C_VEL
LIN {X 0,Y 158.908,Z 579.853,A -85,B 0,C 180,E1 -23848.102,E2 -23848.102} C_VEL
LIN {X 0,Y 158.854,Z 585.239,A -85,B 0,C 180,E1 -23851.27,E2 -23851.27} C_VEL
LIN {X 0,Y 158.193,Z 588.539,A -85,B 0,C 180,E1 -23853.824,E2 -23853.824} C_VEL
LIN {X 0,Y 157.312,Z 592.469,A -85,B 0,C 180,E1 -23857.705,E2 -23857.705} C_VEL
LIN {X 0,Y 157.175,Z 596.315,A -85,B 0,C 180,E1 -23862.922,E2 -23862.922} C_VEL
LIN {X 0,Y 158.743,Z 598.891,A -85,B 0,C 180,E1 -23868.057,E2 -23868.057} C_VEL
LIN {X 0,Y 160.83,Z 599.943,A -85,B 0,C 180,E1 -23871.524,E2 -23871.524} C_VEL
LIN {X 0,Y 161.795,Z 600.253,A -85,B 0,C 180,E1 -23873.592,E2 -23873.592} C_VEL
LIN {X 0,Y 163.069,Z 599.703,A -85,B 0,C 180,E1 -23879.865,E2 -23879.865} C_VEL
LIN {X 0,Y 164.782,Z 599.367,A -85,B 0,C 180,E1 -23881.828,E2 -23881.828} C_VEL
LIN {X 0,Y 165.659,Z 599.243,A -85,B 0,C 180,E1 -23882.435,E2 -23882.435} C_VEL
LIN {X 0,Y 170.626,Z 598.444,A -85,B 0,C 180,E1 -23885.218,E2 -23885.218} C_VEL
LIN {X 0,Y 179.131,Z 596.267,A -85,B 0,C 180,E1 -23888.887,E2 -23888.887} C_VEL
LIN {X 0,Y 188.643,Z 592.898,A -85,B 0,C 180,E1 -23892.116,E2 -23892.116} C_VEL
LIN {X 0,Y 199.073,Z 588.263,A -85,B 0,C 180,E1 -23894.919,E2 -23894.919} C_VEL
LIN {X 0,Y 207.946,Z 583.621,A -85,B 0,C 180,E1 -23896.854,E2 -23896.854} C_VEL
LIN {X 0,Y 207.836,Z 583.497,A -85,B 0,C 180,E1 -23897.444,E2 -23897.444} C_VEL
LIN {X 0,Y 197.318,Z 587.355,A -85,B 0,C 180,E1 -23900.125,E2 -23900.125} C_VEL
LIN {X 0,Y 187.527,Z 589.798,A -85,B 0,C 180,E1 -23903.156,E2 -23903.156} C_VEL
LIN {X 0,Y 178.566,Z 590.9,A -85,B 0,C 180,E1 -23906.563,E2 -23906.563} C_VEL
LIN {X 0,Y 170.595,Z 590.682,A -85,B 0,C 180,E1 -23910.372,E2 -23910.372} C_VEL
LIN {X 0,Y 163.743,Z 589.115,A -85,B 0,C 180,E1 -23914.582,E2 -23914.582} C_VEL
LIN {X 0,Y 158.115,Z 586.22,A -85,B 0,C 180,E1 -23919.17,E2 -23919.17} C_VEL
LIN {X 0,Y 153.782,Z 581.965,A -85,B 0,C 180,E1 -23924.085,E2 -23924.085} C_VEL
LIN {X 0,Y 151.165,Z 576.274,A -85,B 0,C 180,E1 -23929.282,E2 -23929.282} C_VEL
LIN {X 0,Y 149.693,Z 569.856,A -85,B 0,C 180,E1 -23933.936,E2 -23933.936} C_VEL
LIN {X 0,Y 149.133,Z 561.924,A -85,B 0,C 180,E1 -23938.65,E2 -23938.65} C_VEL
LIN {X 0,Y 149.32,Z 553.657,A -85,B 0,C 180,E1 -23942.697,E2 -23942.697} C_VEL
LIN {X 0,Y 149.694,Z 543.387,A -85,B 0,C 180,E1 -23946.74,E2 -23946.74} C_VEL
LIN {X 0,Y 150.401,Z 532.35,A -85,B 0,C 180,E1 -23950.299,E2 -23950.299} C_VEL
LIN {X 0,Y 151.288,Z 520.223,A -85,B 0,C 180,E1 -23953.431,E2 -23953.431} C_VEL
LIN {X 0,Y 152.286,Z 507.529,A -85,B 0,C 180,E1 -23956.075,E2 -23956.075} C_VEL
LIN {X 0,Y 153.281,Z 493.075,A -85,B 0,C 180,E1 -23958.374,E2 -23958.374} C_VEL
LIN {X 0,Y 154.12,Z 479.252,A -85,B 0,C 180,E1 -23959.999,E2 -23959.999} C_VEL
LIN {X 0,Y 157.053,Z 414.007,A -85,B 0,C 180,E1 -23965.776,E2 -23965.776} C_VEL
LIN {X 0,Y 151.233,Z 391.757,A -85,B 0,C 180,E1 -23967.833,E2 -23967.833} C_VEL
LIN {X 0,Y 150.427,Z 387.748,A -85,B 0,C 180,E1 -23968.279,E2 -23968.279} C_VEL
LIN {X 0,Y 150.197,Z 387.771,A -85,B 0,C 180,E1 -23974.16,E2 -23974.16} C_VEL
LIN {X 0,Y 150.178,Z 387.777,A -85,B 0,C 180,E1 -23977.471,E2 -23977.471} C_VEL
LIN {X 0,Y 150.142,Z 387.776,A -85,B 0,C 180,E1 -23981.497,E2 -23981.497} C_VEL
LIN {X 0,Y 150.131,Z 387.783,A -85,B 0,C 180,E1 -23985.393,E2 -23985.393} C_VEL
LIN {X 0,Y 150.16,Z 387.776,A -85,B 0,C 180,E1 -23989.058,E2 -23989.058} C_VEL
LIN {X 0,Y 150.22,Z 387.772,A -85,B 0,C 180,E1 -23992.687,E2 -23992.687} C_VEL
LIN {X 0,Y 150.223,Z 387.77,A -85,B 0,C 180,E1 -23997.363,E2 -23997.363} C_VEL
LIN {X 0,Y 150.249,Z 387.769,A -85,B 0,C 180,E1 -24002.715,E2 -24002.715} C_VEL
LIN {X 0,Y 150.354,Z 387.751,A -85,B 0,C 180,E1 -24009.205,E2 -24009.205} C_VEL
LIN {X 0,Y 150.365,Z 387.755,A -85,B 0,C 180,E1 -24013.711,E2 -24013.711} C_VEL
LIN {X 0,Y 150.614,Z 387.721,A -85,B 0,C 180,E1 -24019.24,E2 -24019.24} C_VEL
LIN {X 0,Y 150.707,Z 387.713,A -85,B 0,C 180,E1 -24021.955,E2 -24021.955} C_VEL
LIN {X 0,Y 151.221,Z 387.65,A -85,B 0,C 180,E1 -24029.997,E2 -24029.997} C_VEL
LIN {X 0,Y 150.763,Z 387.706,A -85,B 0,C 180,E1 -24038.036,E2 -24038.036} C_VEL
LIN {X 0,Y 150.634,Z 387.72,A -85,B 0,C 180,E1 -24041.543,E2 -24041.543} C_VEL
LIN {X 0,Y 150.382,Z 387.753,A -85,B 0,C 180,E1 -24046.281,E2 -24046.281} C_VEL
LIN {X 0,Y 150.349,Z 387.752,A -85,B 0,C 180,E1 -24050.789,E2 -24050.789} C_VEL
LIN {X 0,Y 150.241,Z 387.77,A -85,B 0,C 180,E1 -24057.279,E2 -24057.279} C_VEL
LIN {X 0,Y 150.221,Z 387.77,A -85,B 0,C 180,E1 -24062.636,E2 -24062.636} C_VEL
LIN {X 0,Y 150.265,Z 387.767,A -85,B 0,C 180,E1 -24067.442,E2 -24067.442} C_VEL
LIN {X 0,Y 150.231,Z 387.769,A -85,B 0,C 180,E1 -24071.54,E2 -24071.54} C_VEL
LIN {X 0,Y 150.283,Z 387.765,A -85,B 0,C 180,E1 -24075.455,E2 -24075.455} C_VEL
LIN {X 0,Y 150.232,Z 387.765,A -85,B 0,C 180,E1 -24079.086,E2 -24079.086} C_VEL
LIN {X 0,Y 150.266,Z 387.766,A -85,B 0,C 180,E1 -24082.659,E2 -24082.659} C_VEL
LIN {X 0,Y 150.218,Z 387.767,A -85,B 0,C 180,E1 -24087.36,E2 -24087.36} C_VEL
LIN {X 0,Y 150.237,Z 387.769,A -85,B 0,C 180,E1 -24092.716,E2 -24092.716} C_VEL
LIN {X 0,Y 150.343,Z 387.757,A -85,B 0,C 180,E1 -24099.207,E2 -24099.207} C_VEL
LIN {X 0,Y 150.36,Z 387.75,A -85,B 0,C 180,E1 -24103.713,E2 -24103.713} C_VEL
LIN {X 0,Y 150.681,Z 387.716,A -85,B 0,C 180,E1 -24109.248,E2 -24109.248} C_VEL
LIN {X 0,Y 150.755,Z 387.702,A -85,B 0,C 180,E1 -24111.961,E2 -24111.961} C_VEL
LIN {X 0,Y 151.212,Z 387.646,A -85,B 0,C 180,E1 -24120,E2 -24120} C_VEL
LIN {X 0,Y 150.755,Z 387.704,A -85,B 0,C 180,E1 -24128.04,E2 -24128.04} C_VEL
LIN {X 0,Y 150.627,Z 387.717,A -85,B 0,C 180,E1 -24131.547,E2 -24131.547} C_VEL
LIN {X 0,Y 150.383,Z 387.751,A -85,B 0,C 180,E1 -24136.285,E2 -24136.285} C_VEL
LIN {X 0,Y 150.345,Z 387.752,A -85,B 0,C 180,E1 -24140.795,E2 -24140.795} C_VEL
LIN {X 0,Y 150.237,Z 387.767,A -85,B 0,C 180,E1 -24147.284,E2 -24147.284} C_VEL
LIN {X 0,Y 150.212,Z 387.773,A -85,B 0,C 180,E1 -24152.636,E2 -24152.636} C_VEL
LIN {X 0,Y 150.233,Z 387.766,A -85,B 0,C 180,E1 -24157.456,E2 -24157.456} C_VEL
LIN {X 0,Y 150.235,Z 387.771,A -85,B 0,C 180,E1 -24161.546,E2 -24161.546} C_VEL
LIN {X 0,Y 150.285,Z 387.759,A -85,B 0,C 180,E1 -24165.46,E2 -24165.46} C_VEL
LIN {X 0,Y 150.384,Z 387.751,A -85,B 0,C 180,E1 -24172.606,E2 -24172.606} C_VEL
LIN {X 0,Y 150.681,Z 387.801,A -85,B 0,C 180,E1 -24175.767,E2 -24175.767} C_VEL
LIN {X 0,Y 152.61,Z 396.386,A -85,B 0,C 180,E1 -24180.256,E2 -24180.256} C_VEL
LIN {X 0,Y 153.538,Z 402.725,A -85,B 0,C 180,E1 -24180.828,E2 -24180.828} C_VEL
LIN {X 0,Y 153.974,Z 427.334,A -85,B 0,C 180,E1 -24182.986,E2 -24182.986} C_VEL
LIN {X 0,Y 156.357,Z 460.025,A -85,B 0,C 180,E1 -24185.855,E2 -24185.855} C_VEL
LIN {X 0,Y 154.522,Z 507.258,A -85,B 0,C 180,E1 -24190.232,E2 -24190.232} C_VEL
LIN {X 0,Y 153.926,Z 518.646,A -85,B 0,C 180,E1 -24191.709,E2 -24191.709} C_VEL
LIN {X 0,Y 153.15,Z 530.405,A -85,B 0,C 180,E1 -24193.679,E2 -24193.679} C_VEL
LIN {X 0,Y 152.514,Z 542.651,A -85,B 0,C 180,E1 -24196.292,E2 -24196.292} C_VEL
LIN {X 0,Y 151.941,Z 554.062,A -85,B 0,C 180,E1 -24199.341,E2 -24199.341} C_VEL
LIN {X 0,Y 151.814,Z 562.348,A -85,B 0,C 180,E1 -24202.02,E2 -24202.02} C_VEL
LIN {X 0,Y 151.876,Z 570.879,A -85,B 0,C 180,E1 -24205.358,E2 -24205.358} C_VEL
LIN {X 0,Y 152.249,Z 577.94,A -85,B 0,C 180,E1 -24208.681,E2 -24208.681} C_VEL
LIN {X 0,Y 152.251,Z 582.431,A -85,B 0,C 180,E1 -24211.326,E2 -24211.326} C_VEL
LIN {X 0,Y 151.59,Z 585.972,A -85,B 0,C 180,E1 -24213.991,E2 -24213.991} C_VEL
LIN {X 0,Y 150.663,Z 590.132,A -85,B 0,C 180,E1 -24218.048,E2 -24218.048} C_VEL
LIN {X 0,Y 150.504,Z 594.319,A -85,B 0,C 180,E1 -24223.505,E2 -24223.505} C_VEL
LIN {X 0,Y 152.156,Z 597.236,A -85,B 0,C 180,E1 -24228.867,E2 -24228.867} C_VEL
LIN {X 0,Y 155.522,Z 598.977,A -85,B 0,C 180,E1 -24234.001,E2 -24234.001} C_VEL
LIN {X 0,Y 160.403,Z 599.584,A -85,B 0,C 180,E1 -24238.817,E2 -24238.817} C_VEL
LIN {X 0,Y 165.659,Z 599.243,A -85,B 0,C 180,E1 -24242.435,E2 -24242.435} C_VEL
LIN {X 0,Y 168.104,Z 598.811,A -85,B 0,C 180,E1 -24244.276,E2 -24244.276} C_VEL
LIN {X 0,Y 173.906,Z 596.499,A -85,B 0,C 180,E1 -24249.865,E2 -24249.865} C_VEL
LIN {X 0,Y 176.92,Z 595.534,A -85,B 0,C 180,E1 -24251.479,E2 -24251.479} C_VEL
LIN {X 0,Y 178.176,Z 595.145,A -85,B 0,C 180,E1 -24251.951,E2 -24251.951} C_VEL
LIN {X 0,Y 188.691,Z 591.674,A -85,B 0,C 180,E1 -24255.049,E2 -24255.049} C_VEL
LIN {X 0,Y 194.136,Z 589.508,A -85,B 0,C 180,E1 -24256.391,E2 -24256.391} C_VEL
LIN {X 0,Y 197.428,Z 588.022,A -85,B 0,C 180,E1 -24257.44,E2 -24257.44} C_VEL
LIN {X 0,Y 186.957,Z 590.551,A -85,B 0,C 180,E1 -24260.278,E2 -24260.278} C_VEL
LIN {X 0,Y 177.245,Z 591.761,A -85,B 0,C 180,E1 -24263.503,E2 -24263.503} C_VEL
LIN {X 0,Y 168.497,Z 591.672,A -85,B 0,C 180,E1 -24267.164,E2 -24267.164} C_VEL
LIN {X 0,Y 160.776,Z 590.3,A -85,B 0,C 180,E1 -24271.259,E2 -24271.259} C_VEL
LIN {X 0,Y 154.328,Z 587.62,A -85,B 0,C 180,E1 -24275.804,E2 -24275.804} C_VEL
LIN {X 0,Y 149.095,Z 583.586,A -85,B 0,C 180,E1 -24280.733,E2 -24280.733} C_VEL
LIN {X 0,Y 145.453,Z 578.165,A -85,B 0,C 180,E1 -24286.019,E2 -24286.019} C_VEL
LIN {X 0,Y 143.828,Z 573.106,A -85,B 0,C 180,E1 -24290.152,E2 -24290.152} C_VEL
LIN {X 0,Y 142.581,Z 565.863,A -85,B 0,C 180,E1 -24295.051,E2 -24295.051} C_VEL
LIN {X 0,Y 142.333,Z 556.928,A -85,B 0,C 180,E1 -24300,E2 -24300} C_VEL
LIN {X 0,Y 142.52,Z 549.198,A -85,B 0,C 180,E1 -24303.534,E2 -24303.534} C_VEL
LIN {X 0,Y 143.047,Z 537.963,A -85,B 0,C 180,E1 -24307.765,E2 -24307.765} C_VEL
LIN {X 0,Y 143.801,Z 526.323,A -85,B 0,C 180,E1 -24311.273,E2 -24311.273} C_VEL
LIN {X 0,Y 144.795,Z 513.488,A -85,B 0,C 180,E1 -24314.404,E2 -24314.404} C_VEL
LIN {X 0,Y 145.8,Z 499.738,A -85,B 0,C 180,E1 -24316.991,E2 -24316.991} C_VEL
LIN {X 0,Y 146.714,Z 485.302,A -85,B 0,C 180,E1 -24319.046,E2 -24319.046} C_VEL
LIN {X 0,Y 147.825,Z 461.66,A -85,B 0,C 180,E1 -24321.437,E2 -24321.437} C_VEL
LIN {X 0,Y 149.915,Z 414.841,A -85,B 0,C 180,E1 -24325.777,E2 -24325.777} C_VEL
LIN {X 0,Y 144.234,Z 392.847,A -85,B 0,C 180,E1 -24327.888,E2 -24327.888} C_VEL
LIN {X 0,Y 143.406,Z 388.623,A -85,B 0,C 180,E1 -24328.387,E2 -24328.387} C_VEL
LIN {X 0,Y 143.15,Z 388.647,A -85,B 0,C 180,E1 -24333.418,E2 -24333.418} C_VEL
LIN {X 0,Y 143.061,Z 388.663,A -85,B 0,C 180,E1 -24339.69,E2 -24339.69} C_VEL
LIN {X 0,Y 143.039,Z 388.664,A -85,B 0,C 180,E1 -24343.461,E2 -24343.461} C_VEL
LIN {X 0,Y 143.072,Z 388.662,A -85,B 0,C 180,E1 -24347.462,E2 -24347.462} C_VEL
LIN {X 0,Y 143.111,Z 388.653,A -85,B 0,C 180,E1 -24351.789,E2 -24351.789} C_VEL
LIN {X 0,Y 143.19,Z 388.646,A -85,B 0,C 180,E1 -24357.32,E2 -24357.32} C_VEL
LIN {X 0,Y 143.195,Z 388.647,A -85,B 0,C 180,E1 -24362.06,E2 -24362.06} C_VEL
LIN {X 0,Y 143.28,Z 388.633,A -85,B 0,C 180,E1 -24368.742,E2 -24368.742} C_VEL
LIN {X 0,Y 143.305,Z 388.633,A -85,B 0,C 180,E1 -24372.884,E2 -24372.884} C_VEL
LIN {X 0,Y 143.54,Z 388.603,A -85,B 0,C 180,E1 -24378.703,E2 -24378.703} C_VEL
LIN {X 0,Y 143.629,Z 388.594,A -85,B 0,C 180,E1 -24381.556,E2 -24381.556} C_VEL
LIN {X 0,Y 144.179,Z 388.527,A -85,B 0,C 180,E1 -24389.997,E2 -24389.997} C_VEL
LIN {X 0,Y 143.685,Z 388.587,A -85,B 0,C 180,E1 -24398.435,E2 -24398.435} C_VEL
LIN {X 0,Y 143.57,Z 388.598,A -85,B 0,C 180,E1 -24401.754,E2 -24401.754} C_VEL
LIN {X 0,Y 143.315,Z 388.632,A -85,B 0,C 180,E1 -24407.108,E2 -24407.108} C_VEL
LIN {X 0,Y 143.274,Z 388.633,A -85,B 0,C 180,E1 -24411.251,E2 -24411.251} C_VEL
LIN {X 0,Y 143.187,Z 388.648,A -85,B 0,C 180,E1 -24417.935,E2 -24417.935} C_VEL
LIN {X 0,Y 143.174,Z 388.649,A -85,B 0,C 180,E1 -24423.438,E2 -24423.438} C_VEL
LIN {X 0,Y 143.136,Z 388.649,A -85,B 0,C 180,E1 -24429.661,E2 -24429.661} C_VEL
LIN {X 0,Y 143.177,Z 388.65,A -85,B 0,C 180,E1 -24433.404,E2 -24433.404} C_VEL
LIN {X 0,Y 143.165,Z 388.647,A -85,B 0,C 180,E1 -24437.416,E2 -24437.416} C_VEL
LIN {X 0,Y 143.183,Z 388.65,A -85,B 0,C 180,E1 -24441.747,E2 -24441.747} C_VEL
LIN {X 0,Y 143.186,Z 388.643,A -85,B 0,C 180,E1 -24447.323,E2 -24447.323} C_VEL
LIN {X 0,Y 143.152,Z 388.651,A -85,B 0,C 180,E1 -24453.778,E2 -24453.778} C_VEL
LIN {X 0,Y 143.299,Z 388.635,A -85,B 0,C 180,E1 -24459.922,E2 -24459.922} C_VEL
LIN {X 0,Y 143.364,Z 388.623,A -85,B 0,C 180,E1 -24465.812,E2 -24465.812} C_VEL
LIN {X 0,Y 143.594,Z 388.597,A -85,B 0,C 180,E1 -24468.71,E2 -24468.71} C_VEL
LIN {X 0,Y 143.676,Z 388.585,A -85,B 0,C 180,E1 -24471.562,E2 -24471.562} C_VEL
LIN {X 0,Y 144.171,Z 388.524,A -85,B 0,C 180,E1 -24480,E2 -24480} C_VEL
LIN {X 0,Y 143.677,Z 388.586,A -85,B 0,C 180,E1 -24488.439,E2 -24488.439} C_VEL
LIN {X 0,Y 143.563,Z 388.598,A -85,B 0,C 180,E1 -24491.759,E2 -24491.759} C_VEL
LIN {X 0,Y 143.315,Z 388.633,A -85,B 0,C 180,E1 -24497.112,E2 -24497.112} C_VEL
LIN {X 0,Y 143.27,Z 388.635,A -85,B 0,C 180,E1 -24501.257,E2 -24501.257} C_VEL
LIN {X 0,Y 143.183,Z 388.643,A -85,B 0,C 180,E1 -24507.939,E2 -24507.939} C_VEL
LIN {X 0,Y 143.163,Z 388.652,A -85,B 0,C 180,E1 -24513.438,E2 -24513.438} C_VEL
LIN {X 0,Y 143.128,Z 388.656,A -85,B 0,C 180,E1 -24519.669,E2 -24519.669} C_VEL
LIN {X 0,Y 143.179,Z 388.649,A -85,B 0,C 180,E1 -24523.409,E2 -24523.409} C_VEL
LIN {X 0,Y 143.168,Z 388.648,A -85,B 0,C 180,E1 -24527.421,E2 -24527.421} C_VEL
LIN {X 0,Y 143.575,Z 388.593,A -85,B 0,C 180,E1 -24535.214,E2 -24535.214} C_VEL
LIN {X 0,Y 143.699,Z 388.697,A -85,B 0,C 180,E1 -24536.122,E2 -24536.122} C_VEL
LIN {X 0,Y 145.313,Z 395.785,A -85,B 0,C 180,E1 -24540.023,E2 -24540.023} C_VEL
LIN {X 0,Y 146.464,Z 403.332,A -85,B 0,C 180,E1 -24540.749,E2 -24540.749} C_VEL
LIN {X 0,Y 146.867,Z 427.322,A -85,B 0,C 180,E1 -24542.966,E2 -24542.966} C_VEL
LIN {X 0,Y 149.265,Z 459.607,A -85,B 0,C 180,E1 -24545.951,E2 -24545.951} C_VEL
LIN {X 0,Y 147.517,Z 506.946,A -85,B 0,C 180,E1 -24550.613,E2 -24550.613} C_VEL
LIN {X 0,Y 146.93,Z 518.735,A -85,B 0,C 180,E1 -24552.25,E2 -24552.25} C_VEL
LIN {X 0,Y 146.137,Z 531.894,A -85,B 0,C 180,E1 -24554.648,E2 -24554.648} C_VEL
LIN {X 0,Y 145.563,Z 543.932,A -85,B 0,C 180,E1 -24557.455,E2 -24557.455} C_VEL
LIN {X 0,Y 145.153,Z 555.765,A -85,B 0,C 180,E1 -24560.95,E2 -24560.95} C_VEL
LIN {X 0,Y 145.148,Z 565.379,A -85,B 0,C 180,E1 -24564.446,E2 -24564.446} C_VEL
LIN {X 0,Y 145.591,Z 574.569,A -85,B 0,C 180,E1 -24568.62,E2 -24568.62} C_VEL
LIN {X 0,Y 145.685,Z 579.453,A -85,B 0,C 180,E1 -24571.385,E2 -24571.385} C_VEL
LIN {X 0,Y 145.084,Z 583.188,A -85,B 0,C 180,E1 -24574.17,E2 -24574.17} C_VEL
LIN {X 0,Y 144.068,Z 587.631,A -85,B 0,C 180,E1 -24578.419,E2 -24578.419} C_VEL
LIN {X 0,Y 143.93,Z 592.136,A -85,B 0,C 180,E1 -24584.135,E2 -24584.135} C_VEL
LIN {X 0,Y 145.666,Z 595.389,A -85,B 0,C 180,E1 -24589.742,E2 -24589.742} C_VEL
LIN {X 0,Y 149.176,Z 597.484,A -85,B 0,C 180,E1 -24595.091,E2 -24595.091} C_VEL
LIN {X 0,Y 154.301,Z 598.488,A -85,B 0,C 180,E1 -24600.071,E2 -24600.071} C_VEL
LIN {X 0,Y 161.045,Z 598.444,A -85,B 0,C 180,E1 -24604.567,E2 -24604.567} C_VEL
LIN {X 0,Y 169.165,Z 597.32,A -85,B 0,C 180,E1 -24608.552,E2 -24608.552} C_VEL
LIN {X 0,Y 178.176,Z 595.145,A -85,B 0,C 180,E1 -24611.951,E2 -24611.951} C_VEL
LIN {X 0,Y 179.431,Z 594.697,A -85,B 0,C 180,E1 -24612.688,E2 -24612.688} C_VEL
LIN {X 0,Y 180.807,Z 593.374,A -85,B 0,C 180,E1 -24615.538,E2 -24615.538} C_VEL
LIN {X 0,Y 182.241,Z 592.815,A -85,B 0,C 180,E1 -24616.213,E2 -24616.213} C_VEL
LIN {X 0,Y 186.972,Z 591.351,A -85,B 0,C 180,E1 -24617.422,E2 -24617.422} C_VEL
LIN {X 0,Y 176.562,Z 592.643,A -85,B 0,C 180,E1 -24620.44,E2 -24620.44} C_VEL
LIN {X 0,Y 166.995,Z 592.663,A -85,B 0,C 180,E1 -24623.9,E2 -24623.9} C_VEL
LIN {X 0,Y 158.457,Z 591.417,A -85,B 0,C 180,E1 -24627.843,E2 -24627.843} C_VEL
LIN {X 0,Y 151.061,Z 588.911,A -85,B 0,C 180,E1 -24632.274,E2 -24632.274} C_VEL
LIN {X 0,Y 144.974,Z 585.117,A -85,B 0,C 180,E1 -24637.181,E2 -24637.181} C_VEL
LIN {X 0,Y 140.354,Z 579.929,A -85,B 0,C 180,E1 -24642.516,E2 -24642.516} C_VEL
LIN {X 0,Y 137.522,Z 573.325,A -85,B 0,C 180,E1 -24648.204,E2 -24648.204} C_VEL
LIN {X 0,Y 136.015,Z 566.088,A -85,B 0,C 180,E1 -24653.323,E2 -24653.323} C_VEL
LIN {X 0,Y 135.506,Z 557.144,A -85,B 0,C 180,E1 -24658.514,E2 -24658.514} C_VEL
LIN {X 0,Y 135.731,Z 549.517,A -85,B 0,C 180,E1 -24662.225,E2 -24662.225} C_VEL
LIN {X 0,Y 136.079,Z 538.33,A -85,B 0,C 180,E1 -24666.673,E2 -24666.673} C_VEL
LIN {X 0,Y 136.786,Z 526.955,A -85,B 0,C 180,E1 -24670.319,E2 -24670.319} C_VEL
LIN {X 0,Y 137.722,Z 514.44,A -85,B 0,C 180,E1 -24673.568,E2 -24673.568} C_VEL
LIN {X 0,Y 138.707,Z 500.532,A -85,B 0,C 180,E1 -24676.37,E2 -24676.37} C_VEL
LIN {X 0,Y 139.61,Z 486.442,A -85,B 0,C 180,E1 -24678.528,E2 -24678.528} C_VEL
LIN {X 0,Y 140.602,Z 464.918,A -85,B 0,C 180,E1 -24680.863,E2 -24680.863} C_VEL
LIN {X 0,Y 142.748,Z 415.48,A -85,B 0,C 180,E1 -24685.759,E2 -24685.759} C_VEL
LIN {X 0,Y 137.076,Z 393.25,A -85,B 0,C 180,E1 -24687.977,E2 -24687.977} C_VEL
LIN {X 0,Y 136.368,Z 389.5,A -85,B 0,C 180,E1 -24688.389,E2 -24688.389} C_VEL
LIN {X 0,Y 136.049,Z 389.536,A -85,B 0,C 180,E1 -24694.627,E2 -24694.627} C_VEL
LIN {X 0,Y 136.033,Z 389.538,A -85,B 0,C 180,E1 -24699.194,E2 -24699.194} C_VEL
LIN {X 0,Y 135.984,Z 389.543,A -85,B 0,C 180,E1 -24703.647,E2 -24703.647} C_VEL
LIN {X 0,Y 136.036,Z 389.539,A -85,B 0,C 180,E1 -24707.804,E2 -24707.804} C_VEL
LIN {X 0,Y 136.06,Z 389.531,A -85,B 0,C 180,E1 -24711.691,E2 -24711.691} C_VEL
LIN {X 0,Y 136.095,Z 389.532,A -85,B 0,C 180,E1 -24715.715,E2 -24715.715} C_VEL
LIN {X 0,Y 136.151,Z 389.526,A -85,B 0,C 180,E1 -24722.314,E2 -24722.314} C_VEL
LIN {X 0,Y 136.247,Z 389.509,A -85,B 0,C 180,E1 -24728.83,E2 -24728.83} C_VEL
LIN {X 0,Y 136.271,Z 389.507,A -85,B 0,C 180,E1 -24735.053,E2 -24735.053} C_VEL
LIN {X 0,Y 136.447,Z 389.484,A -85,B 0,C 180,E1 -24738.135,E2 -24738.135} C_VEL
LIN {X 0,Y 136.554,Z 389.474,A -85,B 0,C 180,E1 -24741.115,E2 -24741.115} C_VEL
LIN {X 0,Y 137.136,Z 389.404,A -85,B 0,C 180,E1 -24749.997,E2 -24749.997} C_VEL
LIN {X 0,Y 136.608,Z 389.468,A -85,B 0,C 180,E1 -24758.875,E2 -24758.875} C_VEL
LIN {X 0,Y 136.492,Z 389.478,A -85,B 0,C 180,E1 -24761.954,E2 -24761.954} C_VEL
LIN {X 0,Y 136.25,Z 389.513,A -85,B 0,C 180,E1 -24768.025,E2 -24768.025} C_VEL
LIN {X 0,Y 136.196,Z 389.514,A -85,B 0,C 180,E1 -24771.746,E2 -24771.746} C_VEL
LIN {X 0,Y 136.097,Z 389.529,A -85,B 0,C 180,E1 -24778.614,E2 -24778.614} C_VEL
LIN {X 0,Y 136.088,Z 389.533,A -85,B 0,C 180,E1 -24784.612,E2 -24784.612} C_VEL
LIN {X 0,Y 136.113,Z 389.524,A -85,B 0,C 180,E1 -24789.24,E2 -24789.24} C_VEL
LIN {X 0,Y 136.112,Z 389.531,A -85,B 0,C 180,E1 -24793.708,E2 -24793.708} C_VEL
LIN {X 0,Y 136.116,Z 389.524,A -85,B 0,C 180,E1 -24797.839,E2 -24797.839} C_VEL
LIN {X 0,Y 136.136,Z 389.527,A -85,B 0,C 180,E1 -24801.721,E2 -24801.721} C_VEL
LIN {X 0,Y 136.093,Z 389.528,A -85,B 0,C 180,E1 -24805.71,E2 -24805.71} C_VEL
LIN {X 0,Y 136.139,Z 389.526,A -85,B 0,C 180,E1 -24812.315,E2 -24812.315} C_VEL
LIN {X 0,Y 136.236,Z 389.513,A -85,B 0,C 180,E1 -24818.832,E2 -24818.832} C_VEL
LIN {X 0,Y 136.269,Z 389.503,A -85,B 0,C 180,E1 -24825.056,E2 -24825.056} C_VEL
LIN {X 0,Y 136.492,Z 389.482,A -85,B 0,C 180,E1 -24828.115,E2 -24828.115} C_VEL
LIN {X 0,Y 136.6,Z 389.469,A -85,B 0,C 180,E1 -24831.121,E2 -24831.121} C_VEL
LIN {X 0,Y 137.128,Z 389.401,A -85,B 0,C 180,E1 -24840,E2 -24840} C_VEL
LIN {X 0,Y 136.601,Z 389.468,A -85,B 0,C 180,E1 -24848.879,E2 -24848.879} C_VEL
LIN {X 0,Y 136.485,Z 389.48,A -85,B 0,C 180,E1 -24851.96,E2 -24851.96} C_VEL
LIN {X 0,Y 136.249,Z 389.509,A -85,B 0,C 180,E1 -24858.029,E2 -24858.029} C_VEL
LIN {X 0,Y 136.192,Z 389.519,A -85,B 0,C 180,E1 -24861.751,E2 -24861.751} C_VEL
LIN {X 0,Y 136.093,Z 389.525,A -85,B 0,C 180,E1 -24868.618,E2 -24868.618} C_VEL
LIN {X 0,Y 136.077,Z 389.533,A -85,B 0,C 180,E1 -24874.62,E2 -24874.62} C_VEL
LIN {X 0,Y 136.101,Z 389.529,A -85,B 0,C 180,E1 -24879.24,E2 -24879.24} C_VEL
LIN {X 0,Y 136.114,Z 389.527,A -85,B 0,C 180,E1 -24883.714,E2 -24883.714} C_VEL
LIN {X 0,Y 136.122,Z 389.527,A -85,B 0,C 180,E1 -24887.846,E2 -24887.846} C_VEL
LIN {X 0,Y 136.561,Z 389.466,A -85,B 0,C 180,E1 -24895.525,E2 -24895.525} C_VEL
LIN {X 0,Y 136.756,Z 389.636,A -85,B 0,C 180,E1 -24896.58,E2 -24896.58} C_VEL
LIN {X 0,Y 138.032,Z 395.235,A -85,B 0,C 180,E1 -24899.817,E2 -24899.817} C_VEL
LIN {X 0,Y 139.372,Z 404.082,A -85,B 0,C 180,E1 -24900.717,E2 -24900.717} C_VEL
LIN {X 0,Y 139.819,Z 427.951,A -85,B 0,C 180,E1 -24903.057,E2 -24903.057} C_VEL
LIN {X 0,Y 142.18,Z 460.61,A -85,B 0,C 180,E1 -24906.242,E2 -24906.242} C_VEL
LIN {X 0,Y 140.526,Z 506.34,A -85,B 0,C 180,E1 -24911.035,E2 -24911.035} C_VEL
LIN {X 0,Y 140.022,Z 517.601,A -85,B 0,C 180,E1 -24912.684,E2 -24912.684} C_VEL
LIN {X 0,Y 139.267,Z 530.527,A -85,B 0,C 180,E1 -24915.15,E2 -24915.15} C_VEL
LIN {X 0,Y 138.798,Z 542.098,A -85,B 0,C 180,E1 -24917.947,E2 -24917.947} C_VEL
LIN {X 0,Y 138.477,Z 553.031,A -85,B 0,C 180,E1 -24921.246,E2 -24921.246} C_VEL
LIN {X 0,Y 138.534,Z 562.897,A -85,B 0,C 180,E1 -24924.91,E2 -24924.91} C_VEL
LIN {X 0,Y 138.896,Z 570.933,A -85,B 0,C 180,E1 -24928.554,E2 -24928.554} C_VEL
LIN {X 0,Y 139.156,Z 575.002,A -85,B 0,C 180,E1 -24930.727,E2 -24930.727} C_VEL
LIN {X 0,Y 139.026,Z 578.391,A -85,B 0,C 180,E1 -24932.901,E2 -24932.901} C_VEL
LIN {X 0,Y 137.866,Z 583.489,A -85,B 0,C 180,E1 -24937.325,E2 -24937.325} C_VEL
LIN {X 0,Y 137.319,Z 588.828,A -85,B 0,C 180,E1 -24943.486,E2 -24943.486} C_VEL
LIN {X 0,Y 138.119,Z 591.717,A -85,B 0,C 180,E1 -24947.78,E2 -24947.78} C_VEL
LIN {X 0,Y 140.887,Z 594.733,A -85,B 0,C 180,E1 -24953.524,E2 -24953.524} C_VEL
LIN {X 0,Y 145.411,Z 596.648,A -85,B 0,C 180,E1 -24958.906,E2 -24958.906} C_VEL
LIN {X 0,Y 151.616,Z 597.533,A -85,B 0,C 180,E1 -24963.8,E2 -24963.8} C_VEL
LIN {X 0,Y 159.303,Z 597.396,A -85,B 0,C 180,E1 -24968.147,E2 -24968.147} C_VEL
LIN {X 0,Y 168.323,Z 596.213,A -85,B 0,C 180,E1 -24971.92,E2 -24971.92} C_VEL
LIN {X 0,Y 178.391,Z 593.94,A -85,B 0,C 180,E1 -24975.168,E2 -24975.168} C_VEL
LIN {X 0,Y 182.241,Z 592.815,A -85,B 0,C 180,E1 -24976.213,E2 -24976.213} C_VEL
LIN {X 0,Y 182.606,Z 592.661,A -85,B 0,C 180,E1 -24976.587,E2 -24976.587} C_VEL
LIN {X 0,Y 181.644,Z 592.645,A -85,B 0,C 180,E1 -24977.279,E2 -24977.279} C_VEL
LIN {X 0,Y 178.946,Z 592.933,A -85,B 0,C 180,E1 -24978.069,E2 -24978.069} C_VEL
LIN {X 0,Y 168.57,Z 593.723,A -85,B 0,C 180,E1 -24979.933,E2 -24979.933} C_VEL
LIN {X 0,Y 165.888,Z 593.637,A -85,B 0,C 180,E1 -24980.704,E2 -24980.704} C_VEL
LIN {X 0,Y 156.795,Z 592.514,A -85,B 0,C 180,E1 -24984.359,E2 -24984.359} C_VEL
LIN {X 0,Y 148.503,Z 590.139,A -85,B 0,C 180,E1 -24988.628,E2 -24988.628} C_VEL
LIN {X 0,Y 141.558,Z 586.525,A -85,B 0,C 180,E1 -24993.459,E2 -24993.459} C_VEL
LIN {X 0,Y 135.912,Z 581.592,A -85,B 0,C 180,E1 -24998.778,E2 -24998.778} C_VEL
LIN {X 0,Y 132.026,Z 575.229,A -85,B 0,C 180,E1 -25004.564,E2 -25004.564} C_VEL
LIN {X 0,Y 130.045,Z 568.391,A -85,B 0,C 180,E1 -25009.884,E2 -25009.884} C_VEL
LIN {X 0,Y 128.935,Z 559.99,A -85,B 0,C 180,E1 -25015.31,E2 -25015.31} C_VEL
LIN {X 0,Y 128.876,Z 551.3,A -85,B 0,C 180,E1 -25020,E2 -25020} C_VEL
LIN {X 0,Y 129.047,Z 542.54,A -85,B 0,C 180,E1 -25023.903,E2 -25023.903} C_VEL
LIN {X 0,Y 129.6,Z 530.799,A -85,B 0,C 180,E1 -25028.183,E2 -25028.183} C_VEL
LIN {X 0,Y 130.344,Z 518.983,A -85,B 0,C 180,E1 -25031.665,E2 -25031.665} C_VEL
LIN {X 0,Y 131.235,Z 506.935,A -85,B 0,C 180,E1 -25034.512,E2 -25034.512} C_VEL
LIN {X 0,Y 132.13,Z 493.118,A -85,B 0,C 180,E1 -25037.07,E2 -25037.07} C_VEL
LIN {X 0,Y 132.942,Z 478.96,A -85,B 0,C 180,E1 -25038.993,E2 -25038.993} C_VEL
LIN {X 0,Y 134.337,Z 441.906,A -85,B 0,C 180,E1 -25043,E2 -25043} C_VEL
LIN {X 0,Y 135.622,Z 416.327,A -85,B 0,C 180,E1 -25045.666,E2 -25045.666} C_VEL
LIN {X 0,Y 130.052,Z 394.304,A -85,B 0,C 180,E1 -25047.964,E2 -25047.964} C_VEL
LIN {X 0,Y 129.305,Z 390.379,A -85,B 0,C 180,E1 -25048.443,E2 -25048.443} C_VEL
LIN {X 0,Y 128.965,Z 390.418,A -85,B 0,C 180,E1 -25055.166,E2 -25055.166} C_VEL
LIN {X 0,Y 128.929,Z 390.418,A -85,B 0,C 180,E1 -25060.853,E2 -25060.853} C_VEL
LIN {X 0,Y 128.923,Z 390.425,A -85,B 0,C 180,E1 -25065.127,E2 -25065.127} C_VEL
LIN {X 0,Y 128.962,Z 390.416,A -85,B 0,C 180,E1 -25069.725,E2 -25069.725} C_VEL
LIN {X 0,Y 128.997,Z 390.416,A -85,B 0,C 180,E1 -25074.808,E2 -25074.808} C_VEL
LIN {X 0,Y 129.038,Z 390.408,A -85,B 0,C 180,E1 -25080.644,E2 -25080.644} C_VEL
LIN {X 0,Y 129.112,Z 390.396,A -85,B 0,C 180,E1 -25087.599,E2 -25087.599} C_VEL
LIN {X 0,Y 129.157,Z 390.395,A -85,B 0,C 180,E1 -25090.941,E2 -25090.941} C_VEL
LIN {X 0,Y 129.368,Z 390.364,A -85,B 0,C 180,E1 -25097.919,E2 -25097.919} C_VEL
LIN {X 0,Y 129.479,Z 390.356,A -85,B 0,C 180,E1 -25100.625,E2 -25100.625} C_VEL
LIN {X 0,Y 130.091,Z 390.282,A -85,B 0,C 180,E1 -25109.996,E2 -25109.996} C_VEL
LIN {X 0,Y 129.53,Z 390.35,A -85,B 0,C 180,E1 -25119.364,E2 -25119.364} C_VEL
LIN {X 0,Y 129.393,Z 390.36,A -85,B 0,C 180,E1 -25122.544,E2 -25122.544} C_VEL
LIN {X 0,Y 129.158,Z 390.395,A -85,B 0,C 180,E1 -25129.052,E2 -25129.052} C_VEL
LIN {X 0,Y 129.106,Z 390.397,A -85,B 0,C 180,E1 -25132.395,E2 -25132.395} C_VEL
LIN {X 0,Y 129.032,Z 390.409,A -85,B 0,C 180,E1 -25139.37,E2 -25139.37} C_VEL
LIN {X 0,Y 129.032,Z 390.412,A -85,B 0,C 180,E1 -25145.214,E2 -25145.214} C_VEL
LIN {X 0,Y 129.048,Z 390.406,A -85,B 0,C 180,E1 -25150.803,E2 -25150.803} C_VEL
LIN {X 0,Y 129.033,Z 390.411,A -85,B 0,C 180,E1 -25155.072,E2 -25155.072} C_VEL
LIN {X 0,Y 129.057,Z 390.404,A -85,B 0,C 180,E1 -25159.669,E2 -25159.669} C_VEL
LIN {X 0,Y 129.03,Z 390.41,A -85,B 0,C 180,E1 -25164.781,E2 -25164.781} C_VEL
LIN {X 0,Y 129.043,Z 390.41,A -85,B 0,C 180,E1 -25170.649,E2 -25170.649} C_VEL
LIN {X 0,Y 129.1,Z 390.401,A -85,B 0,C 180,E1 -25177.727,E2 -25177.727} C_VEL
LIN {X 0,Y 129.147,Z 390.397,A -85,B 0,C 180,E1 -25180.943,E2 -25180.943} C_VEL
LIN {X 0,Y 129.41,Z 390.366,A -85,B 0,C 180,E1 -25187.816,E2 -25187.816} C_VEL
LIN {X 0,Y 129.522,Z 390.349,A -85,B 0,C 180,E1 -25190.632,E2 -25190.632} C_VEL
LIN {X 0,Y 130.083,Z 390.278,A -85,B 0,C 180,E1 -25200,E2 -25200} C_VEL
LIN {X 0,Y 129.523,Z 390.347,A -85,B 0,C 180,E1 -25209.369,E2 -25209.369} C_VEL
LIN {X 0,Y 129.387,Z 390.364,A -85,B 0,C 180,E1 -25212.549,E2 -25212.549} C_VEL
LIN {X 0,Y 129.156,Z 390.391,A -85,B 0,C 180,E1 -25219.056,E2 -25219.056} C_VEL
LIN {X 0,Y 129.101,Z 390.402,A -85,B 0,C 180,E1 -25222.4,E2 -25222.4} C_VEL
LIN {X 0,Y 129.029,Z 390.407,A -85,B 0,C 180,E1 -25229.376,E2 -25229.376} C_VEL
LIN {X 0,Y 129.022,Z 390.411,A -85,B 0,C 180,E1 -25235.215,E2 -25235.215} C_VEL
LIN {X 0,Y 129.045,Z 390.41,A -85,B 0,C 180,E1 -25240.809,E2 -25240.809} C_VEL
LIN {X 0,Y 129.035,Z 390.406,A -85,B 0,C 180,E1 -25245.077,E2 -25245.077} C_VEL
LIN {X 0,Y 129.08,Z 390.406,A -85,B 0,C 180,E1 -25249.664,E2 -25249.664} C_VEL
LIN {X 0,Y 129.802,Z 390.507,A -85,B 0,C 180,E1 -25257.113,E2 -25257.113} C_VEL
LIN {X 0,Y 130.791,Z 394.814,A -85,B 0,C 180,E1 -25259.686,E2 -25259.686} C_VEL
LIN {X 0,Y 132.262,Z 404.982,A -85,B 0,C 180,E1 -25260.747,E2 -25260.747} C_VEL
LIN {X 0,Y 132.755,Z 428.356,A -85,B 0,C 180,E1 -25263.178,E2 -25263.178} C_VEL
LIN {X 0,Y 135.134,Z 460.008,A -85,B 0,C 180,E1 -25266.438,E2 -25266.438} C_VEL
LIN {X 0,Y 133.579,Z 505.536,A -85,B 0,C 180,E1 -25271.513,E2 -25271.513} C_VEL
LIN {X 0,Y 133.102,Z 516.913,A -85,B 0,C 180,E1 -25273.283,E2 -25273.283} C_VEL
LIN {X 0,Y 132.434,Z 529.389,A -85,B 0,C 180,E1 -25275.796,E2 -25275.796} C_VEL
LIN {X 0,Y 132.022,Z 541.436,A -85,B 0,C 180,E1 -25278.877,E2 -25278.877} C_VEL
LIN {X 0,Y 131.811,Z 552.302,A -85,B 0,C 180,E1 -25282.343,E2 -25282.343} C_VEL
LIN {X 0,Y 132.002,Z 562.063,A -85,B 0,C 180,E1 -25286.188,E2 -25286.188} C_VEL
LIN {X 0,Y 132.547,Z 570.061,A -85,B 0,C 180,E1 -25290.004,E2 -25290.004} C_VEL
LIN {X 0,Y 132.661,Z 575.137,A -85,B 0,C 180,E1 -25293.04,E2 -25293.04} C_VEL
LIN {X 0,Y 131.483,Z 580.547,A -85,B 0,C 180,E1 -25297.683,E2 -25297.683} C_VEL
LIN {X 0,Y 130.861,Z 584.809,A -85,B 0,C 180,E1 -25302.409,E2 -25302.409} C_VEL
LIN {X 0,Y 131.758,Z 589.349,A -85,B 0,C 180,E1 -25308.669,E2 -25308.669} C_VEL
LIN {X 0,Y 134.67,Z 592.717,A -85,B 0,C 180,E1 -25314.68,E2 -25314.68} C_VEL
LIN {X 0,Y 139.386,Z 594.988,A -85,B 0,C 180,E1 -25320.283,E2 -25320.283} C_VEL
LIN {X 0,Y 145.865,Z 596.276,A -85,B 0,C 180,E1 -25325.326,E2 -25325.326} C_VEL
LIN {X 0,Y 153.821,Z 596.571,A -85,B 0,C 180,E1 -25329.77,E2 -25329.77} C_VEL
LIN {X 0,Y 163.118,Z 595.875,A -85,B 0,C 180,E1 -25333.583,E2 -25333.583} C_VEL
LIN {X 0,Y 174.65,Z 593.87,A -85,B 0,C 180,E1 -25337.154,E2 -25337.154} C_VEL
LIN {X 0,Y 174.668,Z 593.642,A -85,B 0,C 180,E1 -25337.895,E2 -25337.895} C_VEL
LIN {X 0,Y 165.888,Z 593.637,A -85,B 0,C 180,E1 -25340.704,E2 -25340.704} C_VEL
LIN {X 0,Y 161.407,Z 593.363,A -85,B 0,C 180,E1 -25342.046,E2 -25342.046} C_VEL
LIN {X 0,Y 153.073,Z 592.415,A -85,B 0,C 180,E1 -25343.972,E2 -25343.972} C_VEL
LIN {X 0,Y 145.133,Z 590.631,A -85,B 0,C 180,E1 -25346.128,E2 -25346.128} C_VEL
LIN {X 0,Y 141.363,Z 589.176,A -85,B 0,C 180,E1 -25347.843,E2 -25347.843} C_VEL
LIN {X 0,Y 135.307,Z 585.642,A -85,B 0,C 180,E1 -25352.129,E2 -25352.129} C_VEL
LIN {X 0,Y 129.452,Z 580.24,A -85,B 0,C 180,E1 -25357.664,E2 -25357.664} C_VEL
LIN {X 0,Y 125.42,Z 573.423,A -85,B 0,C 180,E1 -25363.729,E2 -25363.729} C_VEL
LIN {X 0,Y 123.352,Z 566.136,A -85,B 0,C 180,E1 -25369.329,E2 -25369.329} C_VEL
LIN {X 0,Y 122.253,Z 557.226,A -85,B 0,C 180,E1 -25375.053,E2 -25375.053} C_VEL
LIN {X 0,Y 122.23,Z 548.031,A -85,B 0,C 180,E1 -25380,E2 -25380} C_VEL
LIN {X 0,Y 122.488,Z 536.526,A -85,B 0,C 180,E1 -25384.937,E2 -25384.937} C_VEL
LIN {X 0,Y 123.077,Z 524.722,A -85,B 0,C 180,E1 -25389.034,E2 -25389.034} C_VEL
LIN {X 0,Y 123.961,Z 511.44,A -85,B 0,C 180,E1 -25392.691,E2 -25392.691} C_VEL
LIN {X 0,Y 124.747,Z 499.553,A -85,B 0,C 180,E1 -25395.285,E2 -25395.285} C_VEL
LIN {X 0,Y 125.664,Z 484.143,A -85,B 0,C 180,E1 -25397.811,E2 -25397.811} C_VEL
LIN {X 0,Y 126.978,Z 452.045,A -85,B 0,C 180,E1 -25401.617,E2 -25401.617} C_VEL
LIN {X 0,Y 128.456,Z 416.947,A -85,B 0,C 180,E1 -25405.536,E2 -25405.536} C_VEL
LIN {X 0,Y 122.839,Z 394.542,A -85,B 0,C 180,E1 -25407.997,E2 -25407.997} C_VEL
LIN {X 0,Y 122.26,Z 391.257,A -85,B 0,C 180,E1 -25408.417,E2 -25408.417} C_VEL
LIN {X 0,Y 121.889,Z 391.301,A -85,B 0,C 180,E1 -25416.168,E2 -25416.168} C_VEL
LIN {X 0,Y 121.87,Z 391.297,A -85,B 0,C 180,E1 -25421.432,E2 -25421.432} C_VEL
LIN {X 0,Y 121.889,Z 391.298,A -85,B 0,C 180,E1 -25428.553,E2 -25428.553} C_VEL
LIN {X 0,Y 121.95,Z 391.294,A -85,B 0,C 180,E1 -25434.805,E2 -25434.805} C_VEL
LIN {X 0,Y 121.946,Z 391.287,A -85,B 0,C 180,E1 -25439.823,E2 -25439.823} C_VEL
LIN {X 0,Y 121.987,Z 391.286,A -85,B 0,C 180,E1 -25446.212,E2 -25446.212} C_VEL
LIN {X 0,Y 122.048,Z 391.278,A -85,B 0,C 180,E1 -25449.784,E2 -25449.784} C_VEL
LIN {X 0,Y 122.242,Z 391.25,A -85,B 0,C 180,E1 -25456.701,E2 -25456.701} C_VEL
LIN {X 0,Y 122.409,Z 391.237,A -85,B 0,C 180,E1 -25460.078,E2 -25460.078} C_VEL
LIN {X 0,Y 122.601,Z 391.209,A -85,B 0,C 180,E1 -25466.71,E2 -25466.71} C_VEL
LIN {X 0,Y 123.044,Z 391.159,A -85,B 0,C 180,E1 -25469.996,E2 -25469.996} C_VEL
LIN {X 0,Y 122.457,Z 391.23,A -85,B 0,C 180,E1 -25476.587,E2 -25476.587} C_VEL
LIN {X 0,Y 122.456,Z 391.231,A -85,B 0,C 180,E1 -25479.91,E2 -25479.91} C_VEL
LIN {X 0,Y 122.263,Z 391.248,A -85,B 0,C 180,E1 -25483.289,E2 -25483.289} C_VEL
LIN {X 0,Y 122.047,Z 391.278,A -85,B 0,C 180,E1 -25490.208,E2 -25490.208} C_VEL
LIN {X 0,Y 121.98,Z 391.287,A -85,B 0,C 180,E1 -25493.781,E2 -25493.781} C_VEL
LIN {X 0,Y 121.939,Z 391.288,A -85,B 0,C 180,E1 -25500.171,E2 -25500.171} C_VEL
LIN {X 0,Y 121.975,Z 391.29,A -85,B 0,C 180,E1 -25506.23,E2 -25506.23} C_VEL
LIN {X 0,Y 121.967,Z 391.289,A -85,B 0,C 180,E1 -25511.489,E2 -25511.489} C_VEL
LIN {X 0,Y 121.97,Z 391.285,A -85,B 0,C 180,E1 -25518.504,E2 -25518.504} C_VEL
LIN {X 0,Y 121.981,Z 391.288,A -85,B 0,C 180,E1 -25524.82,E2 -25524.82} C_VEL
LIN {X 0,Y 121.935,Z 391.295,A -85,B 0,C 180,E1 -25529.824,E2 -25529.824} C_VEL
LIN {X 0,Y 121.976,Z 391.285,A -85,B 0,C 180,E1 -25536.214,E2 -25536.214} C_VEL
LIN {X 0,Y 122.039,Z 391.284,A -85,B 0,C 180,E1 -25539.786,E2 -25539.786} C_VEL
LIN {X 0,Y 122.357,Z 391.243,A -85,B 0,C 180,E1 -25547.522,E2 -25547.522} C_VEL
LIN {X 0,Y 122.448,Z 391.231,A -85,B 0,C 180,E1 -25550.085,E2 -25550.085} C_VEL
LIN {X 0,Y 122.604,Z 391.212,A -85,B 0,C 180,E1 -25556.714,E2 -25556.714} C_VEL
LIN {X 0,Y 123.037,Z 391.156,A -85,B 0,C 180,E1 -25560,E2 -25560} C_VEL
LIN {X 0,Y 122.449,Z 391.232,A -85,B 0,C 180,E1 -25566.592,E2 -25566.592} C_VEL
LIN {X 0,Y 122.449,Z 391.226,A -85,B 0,C 180,E1 -25569.915,E2 -25569.915} C_VEL
LIN {X 0,Y 122.258,Z 391.254,A -85,B 0,C 180,E1 -25573.294,E2 -25573.294} C_VEL
LIN {X 0,Y 122.044,Z 391.276,A -85,B 0,C 180,E1 -25580.214,E2 -25580.214} C_VEL
LIN {X 0,Y 121.976,Z 391.291,A -85,B 0,C 180,E1 -25583.787,E2 -25583.787} C_VEL
LIN {X 0,Y 121.935,Z 391.293,A -85,B 0,C 180,E1 -25590.176,E2 -25590.176} C_VEL
LIN {X 0,Y 121.963,Z 391.287,A -85,B 0,C 180,E1 -25596.229,E2 -25596.229} C_VEL
LIN {X 0,Y 121.965,Z 391.293,A -85,B 0,C 180,E1 -25601.494,E2 -25601.494} C_VEL
LIN {X 0,Y 121.982,Z 391.288,A -85,B 0,C 180,E1 -25608.504,E2 -25608.504} C_VEL
LIN {X 0,Y 122.823,Z 391.211,A -85,B 0,C 180,E1 -25617.621,E2 -25617.621} C_VEL
LIN {X 0,Y 123.514,Z 394.158,A -85,B 0,C 180,E1 -25619.512,E2 -25619.512} C_VEL
LIN {X 0,Y 125.171,Z 405.286,A -85,B 0,C 180,E1 -25620.763,E2 -25620.763} C_VEL
LIN {X 0,Y 125.644,Z 428.384,A -85,B 0,C 180,E1 -25623.321,E2 -25623.321} C_VEL
LIN {X 0,Y 128.07,Z 460.044,A -85,B 0,C 180,E1 -25626.774,E2 -25626.774} C_VEL
LIN {X 0,Y 126.66,Z 505.207,A -85,B 0,C 180,E1 -25632.168,E2 -25632.168} C_VEL
LIN {X 0,Y 126.183,Z 517.622,A -85,B 0,C 180,E1 -25634.249,E2 -25634.249} C_VEL
LIN {X 0,Y 125.609,Z 530.335,A -85,B 0,C 180,E1 -25637.071,E2 -25637.071} C_VEL
LIN {X 0,Y 125.273,Z 541.942,A -85,B 0,C 180,E1 -25640.315,E2 -25640.315} C_VEL
LIN {X 0,Y 125.318,Z 553.556,A -85,B 0,C 180,E1 -25644.372,E2 -25644.372} C_VEL
LIN {X 0,Y 125.689,Z 562.846,A -85,B 0,C 180,E1 -25648.402,E2 -25648.402} C_VEL
LIN {X 0,Y 126.259,Z 569.052,A -85,B 0,C 180,E1 -25651.599,E2 -25651.599} C_VEL
LIN {X 0,Y 126.201,Z 572.727,A -85,B 0,C 180,E1 -25653.995,E2 -25653.995} C_VEL
LIN {X 0,Y 125.173,Z 577.42,A -85,B 0,C 180,E1 -25658.073,E2 -25658.073} C_VEL
LIN {X 0,Y 124.554,Z 583.273,A -85,B 0,C 180,E1 -25664.743,E2 -25664.743} C_VEL
LIN {X 0,Y 126.063,Z 587.822,A -85,B 0,C 180,E1 -25671.25,E2 -25671.25} C_VEL
LIN {X 0,Y 128.571,Z 590.514,A -85,B 0,C 180,E1 -25675.935,E2 -25675.935} C_VEL
LIN {X 0,Y 133.501,Z 593.138,A -85,B 0,C 180,E1 -25681.769,E2 -25681.769} C_VEL
LIN {X 0,Y 140.252,Z 594.811,A -85,B 0,C 180,E1 -25686.968,E2 -25686.968} C_VEL
LIN {X 0,Y 148.502,Z 595.535,A -85,B 0,C 180,E1 -25691.499,E2 -25691.499} C_VEL
LIN {X 0,Y 158.081,Z 595.309,A -85,B 0,C 180,E1 -25695.347,E2 -25695.347} C_VEL
LIN {X 0,Y 163.279,Z 594.824,A -85,B 0,C 180,E1 -25697.035,E2 -25697.035} C_VEL
LIN {X 0,Y 163.954,Z 594.531,A -85,B 0,C 180,E1 -25697.948,E2 -25697.948} C_VEL
LIN {X 0,Y 155.762,Z 593.592,A -85,B 0,C 180,E1 -25700.825,E2 -25700.825} C_VEL
LIN {X 0,Y 146.633,Z 591.321,A -85,B 0,C 180,E1 -25704.889,E2 -25704.889} C_VEL
LIN {X 0,Y 141.363,Z 589.176,A -85,B 0,C 180,E1 -25707.843,E2 -25707.843} C_VEL
LIN {X 0,Y 137.817,Z 587.595,A -85,B 0,C 180,E1 -25709.651,E2 -25709.651} C_VEL
LIN {X 0,Y 131.033,Z 584.207,A -85,B 0,C 180,E1 -25712.367,E2 -25712.367} C_VEL
LIN {X 0,Y 124.789,Z 580.129,A -85,B 0,C 180,E1 -25715.314,E2 -25715.314} C_VEL
LIN {X 0,Y 122.199,Z 577.479,A -85,B 0,C 180,E1 -25717.472,E2 -25717.472} C_VEL
LIN {X 0,Y 118.563,Z 570.329,A -85,B 0,C 180,E1 -25723.646,E2 -25723.646} C_VEL
LIN {X 0,Y 116.548,Z 562.374,A -85,B 0,C 180,E1 -25729.577,E2 -25729.577} C_VEL
LIN {X 0,Y 115.63,Z 552.682,A -85,B 0,C 180,E1 -25735.642,E2 -25735.642} C_VEL
LIN {X 0,Y 115.662,Z 544.395,A -85,B 0,C 180,E1 -25740,E2 -25740} C_VEL
LIN {X 0,Y 115.863,Z 533.198,A -85,B 0,C 180,E1 -25744.784,E2 -25744.784} C_VEL
LIN {X 0,Y 116.38,Z 521.99,A -85,B 0,C 180,E1 -25748.683,E2 -25748.683} C_VEL
LIN {X 0,Y 117.151,Z 509.821,A -85,B 0,C 180,E1 -25752.12,E2 -25752.12} C_VEL
LIN {X 0,Y 117.956,Z 496.618,A -85,B 0,C 180,E1 -25755.026,E2 -25755.026} C_VEL
LIN {X 0,Y 118.798,Z 482.256,A -85,B 0,C 180,E1 -25757.4,E2 -25757.4} C_VEL
LIN {X 0,Y 120.024,Z 448.131,A -85,B 0,C 180,E1 -25761.692,E2 -25761.692} C_VEL
LIN {X 0,Y 121.3,Z 417.575,A -85,B 0,C 180,E1 -25765.344,E2 -25765.344} C_VEL
LIN {X 0,Y 115.767,Z 395.221,A -85,B 0,C 180,E1 -25767.92,E2 -25767.92} C_VEL
LIN {X 0,Y 115.224,Z 392.133,A -85,B 0,C 180,E1 -25768.365,E2 -25768.365} C_VEL
LIN {X 0,Y 114.866,Z 392.169,A -85,B 0,C 180,E1 -25773.412,E2 -25773.412} C_VEL
LIN {X 0,Y 114.783,Z 392.187,A -85,B 0,C 180,E1 -25777.755,E2 -25777.755} C_VEL
LIN {X 0,Y 114.785,Z 392.181,A -85,B 0,C 180,E1 -25782.71,E2 -25782.71} C_VEL
LIN {X 0,Y 114.806,Z 392.184,A -85,B 0,C 180,E1 -25787.667,E2 -25787.667} C_VEL
LIN {X 0,Y 114.817,Z 392.182,A -85,B 0,C 180,E1 -25792.724,E2 -25792.724} C_VEL
LIN {X 0,Y 114.873,Z 392.168,A -85,B 0,C 180,E1 -25798.928,E2 -25798.928} C_VEL
LIN {X 0,Y 114.95,Z 392.161,A -85,B 0,C 180,E1 -25806.504,E2 -25806.504} C_VEL
LIN {X 0,Y 115.014,Z 392.159,A -85,B 0,C 180,E1 -25812.206,E2 -25812.206} C_VEL
LIN {X 0,Y 115.254,Z 392.121,A -85,B 0,C 180,E1 -25817.329,E2 -25817.329} C_VEL
LIN {X 0,Y 115.368,Z 392.112,A -85,B 0,C 180,E1 -25822.998,E2 -25822.998} C_VEL
LIN {X 0,Y 115.996,Z 392.037,A -85,B 0,C 180,E1 -25829.996,E2 -25829.996} C_VEL
LIN {X 0,Y 115.398,Z 392.109,A -85,B 0,C 180,E1 -25836.992,E2 -25836.992} C_VEL
LIN {X 0,Y 115.392,Z 392.109,A -85,B 0,C 180,E1 -25840.524,E2 -25840.524} C_VEL
LIN {X 0,Y 115.147,Z 392.136,A -85,B 0,C 180,E1 -25844.127,E2 -25844.127} C_VEL
LIN {X 0,Y 114.979,Z 392.156,A -85,B 0,C 180,E1 -25851.511,E2 -25851.511} C_VEL
LIN {X 0,Y 114.868,Z 392.176,A -85,B 0,C 180,E1 -25855.354,E2 -25855.354} C_VEL
LIN {X 0,Y 114.867,Z 392.168,A -85,B 0,C 180,E1 -25861.067,E2 -25861.067} C_VEL
LIN {X 0,Y 114.889,Z 392.17,A -85,B 0,C 180,E1 -25867.708,E2 -25867.708} C_VEL
LIN {X 0,Y 114.883,Z 392.174,A -85,B 0,C 180,E1 -25872.769,E2 -25872.769} C_VEL
LIN {X 0,Y 114.893,Z 392.167,A -85,B 0,C 180,E1 -25877.711,E2 -25877.711} C_VEL
LIN {X 0,Y 114.895,Z 392.173,A -85,B 0,C 180,E1 -25882.666,E2 -25882.666} C_VEL
LIN {X 0,Y 114.864,Z 392.173,A -85,B 0,C 180,E1 -25888.928,E2 -25888.928} C_VEL
LIN {X 0,Y 114.939,Z 392.161,A -85,B 0,C 180,E1 -25896.506,E2 -25896.506} C_VEL
LIN {X 0,Y 115.006,Z 392.157,A -85,B 0,C 180,E1 -25902.209,E2 -25902.209} C_VEL
LIN {X 0,Y 115.278,Z 392.123,A -85,B 0,C 180,E1 -25907.257,E2 -25907.257} C_VEL
LIN {X 0,Y 115.385,Z 392.113,A -85,B 0,C 180,E1 -25909.472,E2 -25909.472} C_VEL
LIN {X 0,Y 115.53,Z 392.093,A -85,B 0,C 180,E1 -25916.513,E2 -25916.513} C_VEL
LIN {X 0,Y 115.989,Z 392.034,A -85,B 0,C 180,E1 -25920,E2 -25920} C_VEL
LIN {X 0,Y 115.39,Z 392.112,A -85,B 0,C 180,E1 -25926.997,E2 -25926.997} C_VEL
LIN {X 0,Y 115.385,Z 392.105,A -85,B 0,C 180,E1 -25930.529,E2 -25930.529} C_VEL
LIN {X 0,Y 115.142,Z 392.142,A -85,B 0,C 180,E1 -25934.132,E2 -25934.132} C_VEL
LIN {X 0,Y 114.975,Z 392.159,A -85,B 0,C 180,E1 -25941.516,E2 -25941.516} C_VEL
LIN {X 0,Y 114.864,Z 392.177,A -85,B 0,C 180,E1 -25945.36,E2 -25945.36} C_VEL
LIN {X 0,Y 114.863,Z 392.175,A -85,B 0,C 180,E1 -25951.071,E2 -25951.071} C_VEL
LIN {X 0,Y 114.884,Z 392.168,A -85,B 0,C 180,E1 -25957.717,E2 -25957.717} C_VEL
LIN {X 0,Y 114.883,Z 392.175,A -85,B 0,C 180,E1 -25962.775,E2 -25962.775} C_VEL
LIN {X 0,Y 114.903,Z 392.169,A -85,B 0,C 180,E1 -25967.722,E2 -25967.722} C_VEL
LIN {X 0,Y 115.605,Z 392.079,A -85,B 0,C 180,E1 -25976.834,E2 -25976.834} C_VEL
LIN {X 0,Y 115.905,Z 392.114,A -85,B 0,C 180,E1 -25978.402,E2 -25978.402} C_VEL
LIN {X 0,Y 116.282,Z 393.762,A -85,B 0,C 180,E1 -25979.46,E2 -25979.46} C_VEL
LIN {X 0,Y 118.07,Z 405.654,A -85,B 0,C 180,E1 -25980.848,E2 -25980.848} C_VEL
LIN {X 0,Y 118.694,Z 430.158,A -85,B 0,C 180,E1 -25983.735,E2 -25983.735} C_VEL
LIN {X 0,Y 121.035,Z 459.71,A -85,B 0,C 180,E1 -25987.156,E2 -25987.156} C_VEL
LIN {X 0,Y 119.778,Z 504.839,A -85,B 0,C 180,E1 -25992.944,E2 -25992.944} C_VEL
LIN {X 0,Y 119.324,Z 517.789,A -85,B 0,C 180,E1 -25995.29,E2 -25995.29} C_VEL
LIN {X 0,Y 118.866,Z 531.061,A -85,B 0,C 180,E1 -25998.494,E2 -25998.494} C_VEL
LIN {X 0,Y 118.643,Z 542.253,A -85,B 0,C 180,E1 -26001.916,E2 -26001.916} C_VEL
LIN {X 0,Y 118.923,Z 553.581,A -85,B 0,C 180,E1 -26006.192,E2 -26006.192} C_VEL
LIN {X 0,Y 119.586,Z 563.286,A -85,B 0,C 180,E1 -26010.761,E2 -26010.761} C_VEL
LIN {X 0,Y 120.014,Z 567.864,A -85,B 0,C 180,E1 -26013.361,E2 -26013.361} C_VEL
LIN {X 0,Y 119.653,Z 571.099,A -85,B 0,C 180,E1 -26015.775,E2 -26015.775} C_VEL
LIN {X 0,Y 118.642,Z 575.756,A -85,B 0,C 180,E1 -26020.24,E2 -26020.24} C_VEL
LIN {X 0,Y 118.521,Z 581.579,A -85,B 0,C 180,E1 -26027.251,E2 -26027.251} C_VEL
LIN {X 0,Y 120.684,Z 586.204,A -85,B 0,C 180,E1 -26034.061,E2 -26034.061} C_VEL
LIN {X 0,Y 124.94,Z 589.715,A -85,B 0,C 180,E1 -26040.419,E2 -26040.419} C_VEL
LIN {X 0,Y 131.052,Z 592.216,A -85,B 0,C 180,E1 -26046.154,E2 -26046.154} C_VEL
LIN {X 0,Y 138.904,Z 593.821,A -85,B 0,C 180,E1 -26051.133,E2 -26051.133} C_VEL
LIN {X 0,Y 148.164,Z 594.511,A -85,B 0,C 180,E1 -26055.362,E2 -26055.362} C_VEL
LIN {X 0,Y 153.224,Z 594.508,A -85,B 0,C 180,E1 -26057.217,E2 -26057.217} C_VEL
LIN {X 0,Y 150.331,Z 593.702,A -85,B 0,C 180,E1 -26059.118,E2 -26059.118} C_VEL
LIN {X 0,Y 140.89,Z 590.925,A -85,B 0,C 180,E1 -26063.23,E2 -26063.23} C_VEL
LIN {X 0,Y 132.686,Z 586.955,A -85,B 0,C 180,E1 -26068.016,E2 -26068.016} C_VEL
LIN {X 0,Y 125.889,Z 581.736,A -85,B 0,C 180,E1 -26073.473,E2 -26073.473} C_VEL
LIN {X 0,Y 122.199,Z 577.479,A -85,B 0,C 180,E1 -26077.472,E2 -26077.472} C_VEL
LIN {X 0,Y 119.928,Z 574.701,A -85,B 0,C 180,E1 -26079.684,E2 -26079.684} C_VEL
LIN {X 0,Y 115.317,Z 569.302,A -85,B 0,C 180,E1 -26083.043,E2 -26083.043} C_VEL
LIN {X 0,Y 111.298,Z 563.286,A -85,B 0,C 180,E1 -26086.52,E2 -26086.52} C_VEL
LIN {X 0,Y 110.051,Z 559.615,A -85,B 0,C 180,E1 -26088.875,E2 -26088.875} C_VEL
LIN {X 0,Y 109.12,Z 549.242,A -85,B 0,C 180,E1 -26095.382,E2 -26095.382} C_VEL
LIN {X 0,Y 109.08,Z 540.328,A -85,B 0,C 180,E1 -26100,E2 -26100} C_VEL
LIN {X 0,Y 109.279,Z 529.467,A -85,B 0,C 180,E1 -26104.611,E2 -26104.611} C_VEL
LIN {X 0,Y 109.717,Z 518.957,A -85,B 0,C 180,E1 -26108.286,E2 -26108.286} C_VEL
LIN {X 0,Y 110.491,Z 506.115,A -85,B 0,C 180,E1 -26111.93,E2 -26111.93} C_VEL
LIN {X 0,Y 111.229,Z 493.796,A -85,B 0,C 180,E1 -26114.639,E2 -26114.639} C_VEL
LIN {X 0,Y 111.983,Z 478.833,A -85,B 0,C 180,E1 -26117.108,E2 -26117.108} C_VEL
LIN {X 0,Y 113.141,Z 442.11,A -85,B 0,C 180,E1 -26122.002,E2 -26122.002} C_VEL
LIN {X 0,Y 114.163,Z 418.239,A -85,B 0,C 180,E1 -26125.072,E2 -26125.072} C_VEL
LIN {X 0,Y 108.7,Z 395.989,A -85,B 0,C 180,E1 -26127.758,E2 -26127.758} C_VEL
LIN {X 0,Y 108.193,Z 393.008,A -85,B 0,C 180,E1 -26128.214,E2 -26128.214} C_VEL
LIN {X 0,Y 107.732,Z 393.064,A -85,B 0,C 180,E1 -26135.953,E2 -26135.953} C_VEL
LIN {X 0,Y 107.682,Z 393.065,A -85,B 0,C 180,E1 -26140.742,E2 -26140.742} C_VEL
LIN {X 0,Y 107.684,Z 393.071,A -85,B 0,C 180,E1 -26145.882,E2 -26145.882} C_VEL
LIN {X 0,Y 107.711,Z 393.062,A -85,B 0,C 180,E1 -26151.534,E2 -26151.534} C_VEL
LIN {X 0,Y 107.811,Z 393.048,A -85,B 0,C 180,E1 -26158.562,E2 -26158.562} C_VEL
LIN {X 0,Y 107.914,Z 393.037,A -85,B 0,C 180,E1 -26166.994,E2 -26166.994} C_VEL
LIN {X 0,Y 108.033,Z 393.024,A -85,B 0,C 180,E1 -26174.913,E2 -26174.913} C_VEL
LIN {X 0,Y 108.255,Z 392.998,A -85,B 0,C 180,E1 -26178.765,E2 -26178.765} C_VEL
LIN {X 0,Y 108.449,Z 392.969,A -85,B 0,C 180,E1 -26186.28,E2 -26186.28} C_VEL
LIN {X 0,Y 108.945,Z 392.915,A -85,B 0,C 180,E1 -26189.996,E2 -26189.996} C_VEL
LIN {X 0,Y 108.34,Z 392.988,A -85,B 0,C 180,E1 -26197.45,E2 -26197.45} C_VEL
LIN {X 0,Y 108.202,Z 392.999,A -85,B 0,C 180,E1 -26203.022,E2 -26203.022} C_VEL
LIN {X 0,Y 107.906,Z 393.042,A -85,B 0,C 180,E1 -26209,E2 -26209} C_VEL
LIN {X 0,Y 107.855,Z 393.048,A -85,B 0,C 180,E1 -26214.181,E2 -26214.181} C_VEL
LIN {X 0,Y 107.799,Z 393.052,A -85,B 0,C 180,E1 -26222.055,E2 -26222.055} C_VEL
LIN {X 0,Y 107.79,Z 393.052,A -85,B 0,C 180,E1 -26228.519,E2 -26228.519} C_VEL
LIN {X 0,Y 107.784,Z 393.057,A -85,B 0,C 180,E1 -26235.821,E2 -26235.821} C_VEL
LIN {X 0,Y 107.791,Z 393.057,A -85,B 0,C 180,E1 -26241.474,E2 -26241.474} C_VEL
LIN {X 0,Y 107.807,Z 393.052,A -85,B 0,C 180,E1 -26248.566,E2 -26248.566} C_VEL
LIN {X 0,Y 107.903,Z 393.038,A -85,B 0,C 180,E1 -26256.996,E2 -26256.996} C_VEL
LIN {X 0,Y 108.03,Z 393.02,A -85,B 0,C 180,E1 -26264.917,E2 -26264.917} C_VEL
LIN {X 0,Y 108.298,Z 392.994,A -85,B 0,C 180,E1 -26268.774,E2 -26268.774} C_VEL
LIN {X 0,Y 108.456,Z 392.974,A -85,B 0,C 180,E1 -26276.285,E2 -26276.285} C_VEL
LIN {X 0,Y 108.94,Z 392.912,A -85,B 0,C 180,E1 -26280,E2 -26280} C_VEL
LIN {X 0,Y 108.333,Z 392.991,A -85,B 0,C 180,E1 -26287.455,E2 -26287.455} C_VEL
LIN {X 0,Y 108.195,Z 393.004,A -85,B 0,C 180,E1 -26293.027,E2 -26293.027} C_VEL
LIN {X 0,Y 107.903,Z 393.038,A -85,B 0,C 180,E1 -26299.006,E2 -26299.006} C_VEL
LIN {X 0,Y 107.851,Z 393.05,A -85,B 0,C 180,E1 -26304.187,E2 -26304.187} C_VEL
LIN {X 0,Y 107.794,Z 393.057,A -85,B 0,C 180,E1 -26312.059,E2 -26312.059} C_VEL
LIN {X 0,Y 107.785,Z 393.053,A -85,B 0,C 180,E1 -26318.523,E2 -26318.523} C_VEL
LIN {X 0,Y 107.79,Z 393.05,A -85,B 0,C 180,E1 -26325.826,E2 -26325.826} C_VEL
LIN {X 0,Y 108.179,Z 393.003,A -85,B 0,C 180,E1 -26334.224,E2 -26334.224} C_VEL
LIN {X 0,Y 109.052,Z 393.059,A -85,B 0,C 180,E1 -26339.362,E2 -26339.362} C_VEL
LIN {X 0,Y 110.967,Z 406.226,A -85,B 0,C 180,E1 -26341.029,E2 -26341.029} C_VEL
LIN {X 0,Y 111.678,Z 430.902,A -85,B 0,C 180,E1 -26344.144,E2 -26344.144} C_VEL
LIN {X 0,Y 113.999,Z 459.735,A -85,B 0,C 180,E1 -26347.697,E2 -26347.697} C_VEL
LIN {X 0,Y 112.945,Z 503.733,A -85,B 0,C 180,E1 -26353.743,E2 -26353.743} C_VEL
LIN {X 0,Y 112.645,Z 515.663,A -85,B 0,C 180,E1 -26356.014,E2 -26356.014} C_VEL
LIN {X 0,Y 112.249,Z 528.384,A -85,B 0,C 180,E1 -26359.178,E2 -26359.178} C_VEL
LIN {X 0,Y 112.155,Z 539.863,A -85,B 0,C 180,E1 -26362.805,E2 -26362.805} C_VEL
LIN {X 0,Y 112.491,Z 550.496,A -85,B 0,C 180,E1 -26366.917,E2 -26366.917} C_VEL
LIN {X 0,Y 113.305,Z 560.661,A -85,B 0,C 180,E1 -26371.814,E2 -26371.814} C_VEL
LIN {X 0,Y 113.812,Z 565.221,A -85,B 0,C 180,E1 -26374.446,E2 -26374.446} C_VEL
LIN {X 0,Y 113.347,Z 568.718,A -85,B 0,C 180,E1 -26377.218,E2 -26377.218} C_VEL
LIN {X 0,Y 112.214,Z 575.557,A -85,B 0,C 180,E1 -26384.512,E2 -26384.512} C_VEL
LIN {X 0,Y 113.317,Z 581.079,A -85,B 0,C 180,E1 -26391.851,E2 -26391.851} C_VEL
LIN {X 0,Y 116.783,Z 585.485,A -85,B 0,C 180,E1 -26398.784,E2 -26398.784} C_VEL
LIN {X 0,Y 122.214,Z 588.817,A -85,B 0,C 180,E1 -26405.108,E2 -26405.108} C_VEL
LIN {X 0,Y 129.54,Z 591.247,A -85,B 0,C 180,E1 -26410.624,E2 -26410.624} C_VEL
LIN {X 0,Y 138.407,Z 592.785,A -85,B 0,C 180,E1 -26415.312,E2 -26415.312} C_VEL
LIN {X 0,Y 143.354,Z 593.239,A -85,B 0,C 180,E1 -26417.344,E2 -26417.344} C_VEL
LIN {X 0,Y 140.049,Z 592.062,A -85,B 0,C 180,E1 -26419.279,E2 -26419.279} C_VEL
LIN {X 0,Y 130.878,Z 588.199,A -85,B 0,C 180,E1 -26423.794,E2 -26423.794} C_VEL
LIN {X 0,Y 123.103,Z 583.136,A -85,B 0,C 180,E1 -26429.081,E2 -26429.081} C_VEL
LIN {X 0,Y 116.792,Z 576.755,A -85,B 0,C 180,E1 -26435.087,E2 -26435.087} C_VEL
LIN {X 0,Y 112.494,Z 569.024,A -85,B 0,C 180,E1 -26441.797,E2 -26441.797} C_VEL
LIN {X 0,Y 110.256,Z 560.811,A -85,B 0,C 180,E1 -26448.043,E2 -26448.043} C_VEL
LIN {X 0,Y 110.051,Z 559.615,A -85,B 0,C 180,E1 -26448.875,E2 -26448.875} C_VEL
LIN {X 0,Y 108.99,Z 555.809,A -85,B 0,C 180,E1 -26451.169,E2 -26451.169} C_VEL
LIN {X 0,Y 107.272,Z 551.609,A -85,B 0,C 180,E1 -26453.211,E2 -26453.211} C_VEL
LIN {X 0,Y 103.642,Z 542.575,A -85,B 0,C 180,E1 -26457.043,E2 -26457.043} C_VEL
LIN {X 0,Y 102.675,Z 537.91,A -85,B 0,C 180,E1 -26459.062,E2 -26459.062} C_VEL
LIN {X 0,Y 102.608,Z 536.362,A -85,B 0,C 180,E1 -26459.767,E2 -26459.767} C_VEL
LIN {X 0,Y 102.848,Z 524.107,A -85,B 0,C 180,E1 -26464.9,E2 -26464.9} C_VEL
LIN {X 0,Y 103.329,Z 512.564,A -85,B 0,C 180,E1 -26468.802,E2 -26468.802} C_VEL
LIN {X 0,Y 104.128,Z 498.942,A -85,B 0,C 180,E1 -26472.423,E2 -26472.423} C_VEL
LIN {X 0,Y 104.789,Z 484.366,A -85,B 0,C 180,E1 -26475.312,E2 -26475.312} C_VEL
LIN {X 0,Y 105.632,Z 460.978,A -85,B 0,C 180,E1 -26478.8,E2 -26478.8} C_VEL
LIN {X 0,Y 107.122,Z 419.364,A -85,B 0,C 180,E1 -26484.65,E2 -26484.65} C_VEL
LIN {X 0,Y 101.759,Z 397.289,A -85,B 0,C 180,E1 -26487.445,E2 -26487.445} C_VEL
LIN {X 0,Y 101.173,Z 393.882,A -85,B 0,C 180,E1 -26488.01,E2 -26488.01} C_VEL
LIN {X 0,Y 100.705,Z 393.934,A -85,B 0,C 180,E1 -26493.938,E2 -26493.938} C_VEL
LIN {X 0,Y 100.642,Z 393.945,A -85,B 0,C 180,E1 -26499.805,E2 -26499.805} C_VEL
LIN {X 0,Y 100.654,Z 393.947,A -85,B 0,C 180,E1 -26505.708,E2 -26505.708} C_VEL
LIN {X 0,Y 100.649,Z 393.94,A -85,B 0,C 180,E1 -26511.059,E2 -26511.059} C_VEL
LIN {X 0,Y 100.704,Z 393.938,A -85,B 0,C 180,E1 -26516.872,E2 -26516.872} C_VEL
LIN {X 0,Y 100.789,Z 393.929,A -85,B 0,C 180,E1 -26525.263,E2 -26525.263} C_VEL
LIN {X 0,Y 100.819,Z 393.922,A -85,B 0,C 180,E1 -26529.597,E2 -26529.597} C_VEL
LIN {X 0,Y 101.104,Z 393.882,A -85,B 0,C 180,E1 -26536.698,E2 -26536.698} C_VEL
LIN {X 0,Y 101.245,Z 393.874,A -85,B 0,C 180,E1 -26542.015,E2 -26542.015} C_VEL
LIN {X 0,Y 101.868,Z 393.797,A -85,B 0,C 180,E1 -26549.995,E2 -26549.995} C_VEL
LIN {X 0,Y 101.279,Z 393.869,A -85,B 0,C 180,E1 -26557.973,E2 -26557.973} C_VEL
LIN {X 0,Y 101.128,Z 393.88,A -85,B 0,C 180,E1 -26563.359,E2 -26563.359} C_VEL
LIN {X 0,Y 100.816,Z 393.922,A -85,B 0,C 180,E1 -26570.394,E2 -26570.394} C_VEL
LIN {X 0,Y 100.771,Z 393.931,A -85,B 0,C 180,E1 -26574.954,E2 -26574.954} C_VEL
LIN {X 0,Y 100.71,Z 393.938,A -85,B 0,C 180,E1 -26583.132,E2 -26583.132} C_VEL
LIN {X 0,Y 100.729,Z 393.93,A -85,B 0,C 180,E1 -26589.872,E2 -26589.872} C_VEL
LIN {X 0,Y 100.749,Z 393.933,A -85,B 0,C 180,E1 -26595.768,E2 -26595.768} C_VEL
LIN {X 0,Y 100.73,Z 393.936,A -85,B 0,C 180,E1 -26601.103,E2 -26601.103} C_VEL
LIN {X 0,Y 100.707,Z 393.932,A -85,B 0,C 180,E1 -26606.861,E2 -26606.861} C_VEL
LIN {X 0,Y 100.778,Z 393.924,A -85,B 0,C 180,E1 -26615.265,E2 -26615.265} C_VEL
LIN {X 0,Y 100.809,Z 393.928,A -85,B 0,C 180,E1 -26619.6,E2 -26619.6} C_VEL
LIN {X 0,Y 101.191,Z 393.88,A -85,B 0,C 180,E1 -26627.974,E2 -26627.974} C_VEL
LIN {X 0,Y 101.271,Z 393.865,A -85,B 0,C 180,E1 -26632.022,E2 -26632.022} C_VEL
LIN {X 0,Y 101.864,Z 393.793,A -85,B 0,C 180,E1 -26640,E2 -26640} C_VEL
LIN {X 0,Y 101.272,Z 393.869,A -85,B 0,C 180,E1 -26647.979,E2 -26647.979} C_VEL
LIN {X 0,Y 101.121,Z 393.886,A -85,B 0,C 180,E1 -26653.365,E2 -26653.365} C_VEL
LIN {X 0,Y 100.812,Z 393.92,A -85,B 0,C 180,E1 -26660.4,E2 -26660.4} C_VEL
LIN {X 0,Y 100.767,Z 393.933,A -85,B 0,C 180,E1 -26664.961,E2 -26664.961} C_VEL
LIN {X 0,Y 100.706,Z 393.941,A -85,B 0,C 180,E1 -26673.137,E2 -26673.137} C_VEL
LIN {X 0,Y 100.726,Z 393.937,A -85,B 0,C 180,E1 -26679.877,E2 -26679.877} C_VEL
LIN {X 0,Y 100.754,Z 393.926,A -85,B 0,C 180,E1 -26685.777,E2 -26685.777} C_VEL
LIN {X 0,Y 100.864,Z 393.921,A -85,B 0,C 180,E1 -26691.17,E2 -26691.17} C_VEL
LIN {X 0,Y 101.952,Z 393.786,A -85,B 0,C 180,E1 -26699.503,E2 -26699.503} C_VEL
LIN {X 0,Y 103.877,Z 406.013,A -85,B 0,C 180,E1 -26701.192,E2 -26701.192} C_VEL
LIN {X 0,Y 104.645,Z 430.942,A -85,B 0,C 180,E1 -26704.572,E2 -26704.572} C_VEL
LIN {X 0,Y 106.986,Z 460.223,A -85,B 0,C 180,E1 -26708.431,E2 -26708.431} C_VEL
LIN {X 0,Y 106.159,Z 503.046,A -85,B 0,C 180,E1 -26714.772,E2 -26714.772} C_VEL
LIN {X 0,Y 105.972,Z 514.364,A -85,B 0,C 180,E1 -26717.071,E2 -26717.071} C_VEL
LIN {X 0,Y 105.685,Z 527.109,A -85,B 0,C 180,E1 -26720.435,E2 -26720.435} C_VEL
LIN {X 0,Y 105.748,Z 538.625,A -85,B 0,C 180,E1 -26724.285,E2 -26724.285} C_VEL
LIN {X 0,Y 106.258,Z 548.88,A -85,B 0,C 180,E1 -26728.48,E2 -26728.48} C_VEL
LIN {X 0,Y 107.044,Z 557.658,A -85,B 0,C 180,E1 -26732.844,E2 -26732.844} C_VEL
LIN {X 0,Y 107.631,Z 561.61,A -85,B 0,C 180,E1 -26735.103,E2 -26735.103} C_VEL
LIN {X 0,Y 107.416,Z 564.745,A -85,B 0,C 180,E1 -26737.523,E2 -26737.523} C_VEL
LIN {X 0,Y 106.383,Z 570.395,A -85,B 0,C 180,E1 -26743.373,E2 -26743.373} C_VEL
LIN {X 0,Y 106.99,Z 576.705,A -85,B 0,C 180,E1 -26751.406,E2 -26751.406} C_VEL
LIN {X 0,Y 109.984,Z 581.526,A -85,B 0,C 180,E1 -26758.641,E2 -26758.641} C_VEL
LIN {X 0,Y 113.723,Z 584.592,A -85,B 0,C 180,E1 -26763.797,E2 -26763.797} C_VEL
LIN {X 0,Y 120.412,Z 587.822,A -85,B 0,C 180,E1 -26769.948,E2 -26769.948} C_VEL
LIN {X 0,Y 128.891,Z 590.188,A -85,B 0,C 180,E1 -26775.146,E2 -26775.146} C_VEL
LIN {X 0,Y 133.659,Z 591.057,A -85,B 0,C 180,E1 -26777.408,E2 -26777.408} C_VEL
LIN {X 0,Y 128.472,Z 588.686,A -85,B 0,C 180,E1 -26780.187,E2 -26780.187} C_VEL
LIN {X 0,Y 119.097,Z 582.998,A -85,B 0,C 180,E1 -26785.902,E2 -26785.902} C_VEL
LIN {X 0,Y 112.154,Z 576.498,A -85,B 0,C 180,E1 -26791.967,E2 -26791.967} C_VEL
LIN {X 0,Y 107.102,Z 568.584,A -85,B 0,C 180,E1 -26798.844,E2 -26798.844} C_VEL
LIN {X 0,Y 104.419,Z 560.363,A -85,B 0,C 180,E1 -26805.38,E2 -26805.38} C_VEL
LIN {X 0,Y 102.928,Z 550.381,A -85,B 0,C 180,E1 -26812.151,E2 -26812.151} C_VEL
LIN {X 0,Y 102.731,Z 541.866,A -85,B 0,C 180,E1 -26817.058,E2 -26817.058} C_VEL
LIN {X 0,Y 102.608,Z 536.362,A -85,B 0,C 180,E1 -26819.767,E2 -26819.767} C_VEL
LIN {X 0,Y 102.055,Z 531.673,A -85,B 0,C 180,E1 -26821.682,E2 -26821.682} C_VEL
LIN {X 0,Y 100.723,Z 526.718,A -85,B 0,C 180,E1 -26823.297,E2 -26823.297} C_VEL
LIN {X 0,Y 97.227,Z 514.442,A -85,B 0,C 180,E1 -26826.668,E2 -26826.668} C_VEL
LIN {X 0,Y 96.807,Z 508.96,A -85,B 0,C 180,E1 -26828.24,E2 -26828.24} C_VEL
LIN {X 0,Y 97.476,Z 496.196,A -85,B 0,C 180,E1 -26831.699,E2 -26831.699} C_VEL
LIN {X 0,Y 98.131,Z 481.417,A -85,B 0,C 180,E1 -26834.649,E2 -26834.649} C_VEL
LIN {X 0,Y 98.982,Z 450.352,A -85,B 0,C 180,E1 -26839.575,E2 -26839.575} C_VEL
LIN {X 0,Y 99.956,Z 419.43,A -85,B 0,C 180,E1 -26844.228,E2 -26844.228} C_VEL
LIN {X 0,Y 94.734,Z 398.154,A -85,B 0,C 180,E1 -26847.087,E2 -26847.087} C_VEL
LIN {X 0,Y 94.15,Z 394.756,A -85,B 0,C 180,E1 -26847.658,E2 -26847.658} C_VEL
LIN {X 0,Y 93.621,Z 394.817,A -85,B 0,C 180,E1 -26854.326,E2 -26854.326} C_VEL
LIN {X 0,Y 93.536,Z 394.826,A -85,B 0,C 180,E1 -26862.549,E2 -26862.549} C_VEL
LIN {X 0,Y 93.548,Z 394.828,A -85,B 0,C 180,E1 -26868.7,E2 -26868.7} C_VEL
LIN {X 0,Y 93.603,Z 394.826,A -85,B 0,C 180,E1 -26875.681,E2 -26875.681} C_VEL
LIN {X 0,Y 93.673,Z 394.817,A -85,B 0,C 180,E1 -26884.2,E2 -26884.2} C_VEL
LIN {X 0,Y 93.695,Z 394.806,A -85,B 0,C 180,E1 -26887.968,E2 -26887.968} C_VEL
LIN {X 0,Y 94.024,Z 394.765,A -85,B 0,C 180,E1 -26896.337,E2 -26896.337} C_VEL
LIN {X 0,Y 94.178,Z 394.754,A -85,B 0,C 180,E1 -26901.412,E2 -26901.412} C_VEL
LIN {X 0,Y 94.794,Z 394.678,A -85,B 0,C 180,E1 -26909.995,E2 -26909.995} C_VEL
LIN {X 0,Y 94.211,Z 394.75,A -85,B 0,C 180,E1 -26918.575,E2 -26918.575} C_VEL
LIN {X 0,Y 94.046,Z 394.762,A -85,B 0,C 180,E1 -26923.717,E2 -26923.717} C_VEL
LIN {X 0,Y 93.691,Z 394.806,A -85,B 0,C 180,E1 -26932.023,E2 -26932.023} C_VEL
LIN {X 0,Y 93.621,Z 394.823,A -85,B 0,C 180,E1 -26936.764,E2 -26936.764} C_VEL
LIN {X 0,Y 93.623,Z 394.823,A -85,B 0,C 180,E1 -26944.338,E2 -26944.338} C_VEL
LIN {X 0,Y 93.646,Z 394.819,A -85,B 0,C 180,E1 -26952.481,E2 -26952.481} C_VEL
LIN {X 0,Y 93.646,Z 394.812,A -85,B 0,C 180,E1 -26958.625,E2 -26958.625} C_VEL
LIN {X 0,Y 93.621,Z 394.817,A -85,B 0,C 180,E1 -26965.655,E2 -26965.655} C_VEL
LIN {X 0,Y 93.662,Z 394.813,A -85,B 0,C 180,E1 -26974.202,E2 -26974.202} C_VEL
LIN {X 0,Y 93.685,Z 394.812,A -85,B 0,C 180,E1 -26977.971,E2 -26977.971} C_VEL
LIN {X 0,Y 94.09,Z 394.762,A -85,B 0,C 180,E1 -26987.051,E2 -26987.051} C_VEL
LIN {X 0,Y 94.203,Z 394.747,A -85,B 0,C 180,E1 -26991.419,E2 -26991.419} C_VEL
LIN {X 0,Y 94.79,Z 394.674,A -85,B 0,C 180,E1 -27000,E2 -27000} C_VEL
LIN {X 0,Y 94.204,Z 394.749,A -85,B 0,C 180,E1 -27008.582,E2 -27008.582} C_VEL
LIN {X 0,Y 94.039,Z 394.77,A -85,B 0,C 180,E1 -27013.723,E2 -27013.723} C_VEL
LIN {X 0,Y 93.688,Z 394.813,A -85,B 0,C 180,E1 -27022.03,E2 -27022.03} C_VEL
LIN {X 0,Y 93.617,Z 394.82,A -85,B 0,C 180,E1 -27026.772,E2 -27026.772} C_VEL
LIN {X 0,Y 93.619,Z 394.822,A -85,B 0,C 180,E1 -27034.343,E2 -27034.343} C_VEL
LIN {X 0,Y 93.647,Z 394.82,A -85,B 0,C 180,E1 -27042.489,E2 -27042.489} C_VEL
LIN {X 0,Y 93.701,Z 394.811,A -85,B 0,C 180,E1 -27048.595,E2 -27048.595} C_VEL
LIN {X 0,Y 94.95,Z 394.717,A -85,B 0,C 180,E1 -27059.9,E2 -27059.9} C_VEL
LIN {X 0,Y 96.801,Z 407.329,A -85,B 0,C 180,E1 -27061.667,E2 -27061.667} C_VEL
LIN {X 0,Y 97.757,Z 432.973,A -85,B 0,C 180,E1 -27065.411,E2 -27065.411} C_VEL
LIN {X 0,Y 100.054,Z 459.612,A -85,B 0,C 180,E1 -27069.16,E2 -27069.16} C_VEL
LIN {X 0,Y 99.453,Z 503.426,A -85,B 0,C 180,E1 -27076.207,E2 -27076.207} C_VEL
LIN {X 0,Y 99.312,Z 514.87,A -85,B 0,C 180,E1 -27078.783,E2 -27078.783} C_VEL
LIN {X 0,Y 99.299,Z 528.517,A -85,B 0,C 180,E1 -27082.787,E2 -27082.787} C_VEL
LIN {X 0,Y 99.571,Z 539.788,A -85,B 0,C 180,E1 -27086.982,E2 -27086.982} C_VEL
LIN {X 0,Y 100.298,Z 548.755,A -85,B 0,C 180,E1 -27091.008,E2 -27091.008} C_VEL
LIN {X 0,Y 101.531,Z 558.15,A -85,B 0,C 180,E1 -27096.13,E2 -27096.13} C_VEL
LIN {X 0,Y 101.589,Z 560.67,A -85,B 0,C 180,E1 -27097.958,E2 -27097.958} C_VEL
LIN {X 0,Y 100.567,Z 566.424,A -85,B 0,C 180,E1 -27103.956,E2 -27103.956} C_VEL
LIN {X 0,Y 101.187,Z 573.079,A -85,B 0,C 180,E1 -27112.463,E2 -27112.463} C_VEL
LIN {X 0,Y 104.446,Z 578.398,A -85,B 0,C 180,E1 -27120.314,E2 -27120.314} C_VEL
LIN {X 0,Y 111.669,Z 583.597,A -85,B 0,C 180,E1 -27129.008,E2 -27129.008} C_VEL
LIN {X 0,Y 119.646,Z 586.758,A -85,B 0,C 180,E1 -27134.825,E2 -27134.825} C_VEL
LIN {X 0,Y 124.229,Z 588.025,A -85,B 0,C 180,E1 -27137.35,E2 -27137.35} C_VEL
LIN {X 0,Y 119.885,Z 585.588,A -85,B 0,C 180,E1 -27139.845,E2 -27139.845} C_VEL
LIN {X 0,Y 111.512,Z 579.573,A -85,B 0,C 180,E1 -27145.443,E2 -27145.443} C_VEL
LIN {X 0,Y 104.692,Z 572.212,A -85,B 0,C 180,E1 -27151.971,E2 -27151.971} C_VEL
LIN {X 0,Y 100.067,Z 563.51,A -85,B 0,C 180,E1 -27159.441,E2 -27159.441} C_VEL
LIN {X 0,Y 97.606,Z 554.294,A -85,B 0,C 180,E1 -27166.466,E2 -27166.466} C_VEL
LIN {X 0,Y 96.514,Z 543.068,A -85,B 0,C 180,E1 -27173.729,E2 -27173.729} C_VEL
LIN {X 0,Y 96.271,Z 534.216,A -85,B 0,C 180,E1 -27178.431,E2 -27178.431} C_VEL
LIN {X 0,Y 96.358,Z 522.278,A -85,B 0,C 180,E1 -27183.659,E2 -27183.659} C_VEL
LIN {X 0,Y 96.807,Z 508.96,A -85,B 0,C 180,E1 -27188.24,E2 -27188.24} C_VEL
LIN {X 0,Y 96.42,Z 503.606,A -85,B 0,C 180,E1 -27189.646,E2 -27189.646} C_VEL
LIN {X 0,Y 94.167,Z 494.42,A -85,B 0,C 180,E1 -27191.327,E2 -27191.327} C_VEL
LIN {X 0,Y 91.846,Z 485.001,A -85,B 0,C 180,E1 -27192.73,E2 -27192.73} C_VEL
LIN {X 0,Y 91.433,Z 479.097,A -85,B 0,C 180,E1 -27193.678,E2 -27193.678} C_VEL
LIN {X 0,Y 92.059,Z 445.927,A -85,B 0,C 180,E1 -27199.366,E2 -27199.366} C_VEL
LIN {X 0,Y 92.914,Z 420.08,A -85,B 0,C 180,E1 -27203.596,E2 -27203.596} C_VEL
LIN {X 0,Y 88.001,Z 400.447,A -85,B 0,C 180,E1 -27206.381,E2 -27206.381} C_VEL
LIN {X 0,Y 87.155,Z 395.628,A -85,B 0,C 180,E1 -27207.256,E2 -27207.256} C_VEL
LIN {X 0,Y 86.53,Z 395.705,A -85,B 0,C 180,E1 -27215.679,E2 -27215.679} C_VEL
LIN {X 0,Y 86.48,Z 395.707,A -85,B 0,C 180,E1 -27222.988,E2 -27222.988} C_VEL
LIN {X 0,Y 86.469,Z 395.707,A -85,B 0,C 180,E1 -27229.435,E2 -27229.435} C_VEL
LIN {X 0,Y 86.547,Z 395.704,A -85,B 0,C 180,E1 -27235.353,E2 -27235.353} C_VEL
LIN {X 0,Y 86.589,Z 395.699,A -85,B 0,C 180,E1 -27243.229,E2 -27243.229} C_VEL
LIN {X 0,Y 86.648,Z 395.691,A -85,B 0,C 180,E1 -27251.063,E2 -27251.063} C_VEL
LIN {X 0,Y 86.933,Z 395.648,A -85,B 0,C 180,E1 -27255.959,E2 -27255.959} C_VEL
LIN {X 0,Y 87.087,Z 395.637,A -85,B 0,C 180,E1 -27260.706,E2 -27260.706} C_VEL
LIN {X 0,Y 87.72,Z 395.559,A -85,B 0,C 180,E1 -27269.995,E2 -27269.995} C_VEL
LIN {X 0,Y 87.117,Z 395.633,A -85,B 0,C 180,E1 -27279.28,E2 -27279.28} C_VEL
LIN {X 0,Y 86.948,Z 395.647,A -85,B 0,C 180,E1 -27284.082,E2 -27284.082} C_VEL
LIN {X 0,Y 86.662,Z 395.689,A -85,B 0,C 180,E1 -27288.923,E2 -27288.923} C_VEL
LIN {X 0,Y 86.582,Z 395.7,A -85,B 0,C 180,E1 -27296.763,E2 -27296.763} C_VEL
LIN {X 0,Y 86.551,Z 395.704,A -85,B 0,C 180,E1 -27305.708,E2 -27305.708} C_VEL
LIN {X 0,Y 86.57,Z 395.701,A -85,B 0,C 180,E1 -27313.06,E2 -27313.06} C_VEL
LIN {X 0,Y 86.567,Z 395.695,A -85,B 0,C 180,E1 -27319.498,E2 -27319.498} C_VEL
LIN {X 0,Y 86.572,Z 395.696,A -85,B 0,C 180,E1 -27325.371,E2 -27325.371} C_VEL
LIN {X 0,Y 86.579,Z 395.699,A -85,B 0,C 180,E1 -27333.23,E2 -27333.23} C_VEL
LIN {X 0,Y 86.655,Z 395.691,A -85,B 0,C 180,E1 -27341.07,E2 -27341.07} C_VEL
LIN {X 0,Y 86.961,Z 395.646,A -85,B 0,C 180,E1 -27345.969,E2 -27345.969} C_VEL
LIN {X 0,Y 87.11,Z 395.633,A -85,B 0,C 180,E1 -27350.715,E2 -27350.715} C_VEL
LIN {X 0,Y 87.718,Z 395.555,A -85,B 0,C 180,E1 -27360.001,E2 -27360.001} C_VEL
LIN {X 0,Y 87.11,Z 395.629,A -85,B 0,C 180,E1 -27369.286,E2 -27369.286} C_VEL
LIN {X 0,Y 86.943,Z 395.655,A -85,B 0,C 180,E1 -27374.089,E2 -27374.089} C_VEL
LIN {X 0,Y 86.581,Z 395.7,A -85,B 0,C 180,E1 -27383.946,E2 -27383.946} C_VEL
LIN {X 0,Y 86.475,Z 395.705,A -85,B 0,C 180,E1 -27389.186,E2 -27389.186} C_VEL
LIN {X 0,Y 86.547,Z 395.699,A -85,B 0,C 180,E1 -27395.714,E2 -27395.714} C_VEL
LIN {X 0,Y 86.593,Z 395.697,A -85,B 0,C 180,E1 -27403.084,E2 -27403.084} C_VEL
LIN {X 0,Y 86.664,Z 395.69,A -85,B 0,C 180,E1 -27409.559,E2 -27409.559} C_VEL
LIN {X 0,Y 87.923,Z 395.533,A -85,B 0,C 180,E1 -27420.281,E2 -27420.281} C_VEL
LIN {X 0,Y 89.76,Z 407.739,A -85,B 0,C 180,E1 -27422.144,E2 -27422.144} C_VEL
LIN {X 0,Y 90.699,Z 432.103,A -85,B 0,C 180,E1 -27426.004,E2 -27426.004} C_VEL
LIN {X 0,Y 93.124,Z 459.493,A -85,B 0,C 180,E1 -27430.152,E2 -27430.152} C_VEL
LIN {X 0,Y 92.853,Z 501.72,A -85,B 0,C 180,E1 -27437.492,E2 -27437.492} C_VEL
LIN {X 0,Y 92.838,Z 513.2,A -85,B 0,C 180,E1 -27440.209,E2 -27440.209} C_VEL
LIN {X 0,Y 92.979,Z 526.46,A -85,B 0,C 180,E1 -27444.31,E2 -27444.31} C_VEL
LIN {X 0,Y 93.517,Z 538.453,A -85,B 0,C 180,E1 -27449.044,E2 -27449.044} C_VEL
LIN {X 0,Y 94.405,Z 547.196,A -85,B 0,C 180,E1 -27453.206,E2 -27453.206} C_VEL
LIN {X 0,Y 95.803,Z 556.269,A -85,B 0,C 180,E1 -27458.442,E2 -27458.442} C_VEL
LIN {X 0,Y 95.478,Z 558.902,A -85,B 0,C 180,E1 -27460.872,E2 -27460.872} C_VEL
LIN {X 0,Y 94.889,Z 566.158,A -85,B 0,C 180,E1 -27469.474,E2 -27469.474} C_VEL
LIN {X 0,Y 96.896,Z 572.154,A -85,B 0,C 180,E1 -27477.813,E2 -27477.813} C_VEL
LIN {X 0,Y 101.792,Z 577.468,A -85,B 0,C 180,E1 -27485.94,E2 -27485.94} C_VEL
LIN {X 0,Y 106.731,Z 580.63,A -85,B 0,C 180,E1 -27491.189,E2 -27491.189} C_VEL
LIN {X 0,Y 115.055,Z 584.159,A -85,B 0,C 180,E1 -27497.145,E2 -27497.145} C_VEL
LIN {X 0,Y 114.705,Z 583.862,A -85,B 0,C 180,E1 -27497.625,E2 -27497.625} C_VEL
LIN {X 0,Y 106.006,Z 577.35,A -85,B 0,C 180,E1 -27503.367,E2 -27503.367} C_VEL
LIN {X 0,Y 98.885,Z 569.503,A -85,B 0,C 180,E1 -27510.164,E2 -27510.164} C_VEL
LIN {X 0,Y 94.049,Z 560.316,A -85,B 0,C 180,E1 -27518.059,E2 -27518.059} C_VEL
LIN {X 0,Y 91.735,Z 552.077,A -85,B 0,C 180,E1 -27524.446,E2 -27524.446} C_VEL
LIN {X 0,Y 90.41,Z 540.495,A -85,B 0,C 180,E1 -27532.181,E2 -27532.181} C_VEL
LIN {X 0,Y 90.024,Z 531.28,A -85,B 0,C 180,E1 -27537.203,E2 -27537.203} C_VEL
LIN {X 0,Y 89.999,Z 520.148,A -85,B 0,C 180,E1 -27542.237,E2 -27542.237} C_VEL
LIN {X 0,Y 90.277,Z 507.477,A -85,B 0,C 180,E1 -27546.814,E2 -27546.814} C_VEL
LIN {X 0,Y 90.86,Z 494.097,A -85,B 0,C 180,E1 -27550.585,E2 -27550.585} C_VEL
LIN {X 0,Y 91.433,Z 479.097,A -85,B 0,C 180,E1 -27553.678,E2 -27553.678} C_VEL
LIN {X 0,Y 90.97,Z 473.383,A -85,B 0,C 180,E1 -27554.562,E2 -27554.562} C_VEL
LIN {X 0,Y 85.752,Z 454.533,A -85,B 0,C 180,E1 -27556.829,E2 -27556.829} C_VEL
LIN {X 0,Y 85.15,Z 448.787,A -85,B 0,C 180,E1 -27557.744,E2 -27557.744} C_VEL
LIN {X 0,Y 85.88,Z 420.746,A -85,B 0,C 180,E1 -27562.784,E2 -27562.784} C_VEL
LIN {X 0,Y 81.039,Z 401.301,A -85,B 0,C 180,E1 -27565.697,E2 -27565.697} C_VEL
LIN {X 0,Y 80.194,Z 396.493,A -85,B 0,C 180,E1 -27566.551,E2 -27566.551} C_VEL
LIN {X 0,Y 79.401,Z 396.594,A -85,B 0,C 180,E1 -27577.183,E2 -27577.183} C_VEL
LIN {X 0,Y 79.391,Z 396.595,A -85,B 0,C 180,E1 -27585.087,E2 -27585.087} C_VEL
LIN {X 0,Y 79.398,Z 396.592,A -85,B 0,C 180,E1 -27592.81,E2 -27592.81} C_VEL
LIN {X 0,Y 79.389,Z 396.589,A -85,B 0,C 180,E1 -27597.91,E2 -27597.91} C_VEL
LIN {X 0,Y 79.529,Z 396.579,A -85,B 0,C 180,E1 -27603.772,E2 -27603.772} C_VEL
LIN {X 0,Y 79.516,Z 396.574,A -85,B 0,C 180,E1 -27609.29,E2 -27609.29} C_VEL
LIN {X 0,Y 79.827,Z 396.535,A -85,B 0,C 180,E1 -27615.567,E2 -27615.567} C_VEL
LIN {X 0,Y 79.97,Z 396.522,A -85,B 0,C 180,E1 -27619.871,E2 -27619.871} C_VEL
LIN {X 0,Y 80.647,Z 396.44,A -85,B 0,C 180,E1 -27629.994,E2 -27629.994} C_VEL
LIN {X 0,Y 79.999,Z 396.518,A -85,B 0,C 180,E1 -27640.113,E2 -27640.113} C_VEL
LIN {X 0,Y 79.764,Z 396.546,A -85,B 0,C 180,E1 -27645.321,E2 -27645.321} C_VEL
LIN {X 0,Y 79.521,Z 396.573,A -85,B 0,C 180,E1 -27650.696,E2 -27650.696} C_VEL
LIN {X 0,Y 79.481,Z 396.583,A -85,B 0,C 180,E1 -27657.844,E2 -27657.844} C_VEL
LIN {X 0,Y 79.461,Z 396.584,A -85,B 0,C 180,E1 -27667.25,E2 -27667.25} C_VEL
LIN {X 0,Y 79.489,Z 396.583,A -85,B 0,C 180,E1 -27675.009,E2 -27675.009} C_VEL
LIN {X 0,Y 79.46,Z 396.587,A -85,B 0,C 180,E1 -27682.742,E2 -27682.742} C_VEL
LIN {X 0,Y 79.478,Z 396.584,A -85,B 0,C 180,E1 -27692.148,E2 -27692.148} C_VEL
LIN {X 0,Y 79.515,Z 396.58,A -85,B 0,C 180,E1 -27699.296,E2 -27699.296} C_VEL
LIN {X 0,Y 79.834,Z 396.532,A -85,B 0,C 180,E1 -27705.524,E2 -27705.524} C_VEL
LIN {X 0,Y 79.992,Z 396.52,A -85,B 0,C 180,E1 -27709.88,E2 -27709.88} C_VEL
LIN {X 0,Y 80.646,Z 396.436,A -85,B 0,C 180,E1 -27720.001,E2 -27720.001} C_VEL
LIN {X 0,Y 79.993,Z 396.513,A -85,B 0,C 180,E1 -27730.121,E2 -27730.121} C_VEL
LIN {X 0,Y 79.755,Z 396.551,A -85,B 0,C 180,E1 -27735.329,E2 -27735.329} C_VEL
LIN {X 0,Y 79.508,Z 396.574,A -85,B 0,C 180,E1 -27740.707,E2 -27740.707} C_VEL
LIN {X 0,Y 79.478,Z 396.576,A -85,B 0,C 180,E1 -27747.851,E2 -27747.851} C_VEL
LIN {X 0,Y 79.458,Z 396.579,A -85,B 0,C 180,E1 -27757.257,E2 -27757.257} C_VEL
LIN {X 0,Y 79.507,Z 396.574,A -85,B 0,C 180,E1 -27765.005,E2 -27765.005} C_VEL
LIN {X 0,Y 79.768,Z 396.546,A -85,B 0,C 180,E1 -27772.464,E2 -27772.464} C_VEL
LIN {X 0,Y 80.935,Z 396.403,A -85,B 0,C 180,E1 -27780.897,E2 -27780.897} C_VEL
LIN {X 0,Y 82.737,Z 407.818,A -85,B 0,C 180,E1 -27782.747,E2 -27782.747} C_VEL
LIN {X 0,Y 83.743,Z 431.933,A -85,B 0,C 180,E1 -27786.895,E2 -27786.895} C_VEL
LIN {X 0,Y 86.292,Z 459.818,A -85,B 0,C 180,E1 -27791.455,E2 -27791.455} C_VEL
LIN {X 0,Y 86.365,Z 501.35,A -85,B 0,C 180,E1 -27799.337,E2 -27799.337} C_VEL
LIN {X 0,Y 86.474,Z 512.834,A -85,B 0,C 180,E1 -27802.316,E2 -27802.316} C_VEL
LIN {X 0,Y 86.849,Z 525.494,A -85,B 0,C 180,E1 -27806.526,E2 -27806.526} C_VEL
LIN {X 0,Y 87.592,Z 536.485,A -85,B 0,C 180,E1 -27811.155,E2 -27811.155} C_VEL
LIN {X 0,Y 88.72,Z 545.523,A -85,B 0,C 180,E1 -27815.688,E2 -27815.688} C_VEL
LIN {X 0,Y 90.019,Z 552.566,A -85,B 0,C 180,E1 -27819.859,E2 -27819.859} C_VEL
LIN {X 0,Y 89.776,Z 555.399,A -85,B 0,C 180,E1 -27822.521,E2 -27822.521} C_VEL
LIN {X 0,Y 89.388,Z 561.927,A -85,B 0,C 180,E1 -27830.485,E2 -27830.485} C_VEL
LIN {X 0,Y 91.747,Z 568.601,A -85,B 0,C 180,E1 -27839.867,E2 -27839.867} C_VEL
LIN {X 0,Y 96.819,Z 574.05,A -85,B 0,C 180,E1 -27848.103,E2 -27848.103} C_VEL
LIN {X 0,Y 106.179,Z 579.479,A -85,B 0,C 180,E1 -27856.733,E2 -27856.733} C_VEL
LIN {X 0,Y 105.038,Z 578.482,A -85,B 0,C 180,E1 -27858.002,E2 -27858.002} C_VEL
LIN {X 0,Y 95.845,Z 569.794,A -85,B 0,C 180,E1 -27865.369,E2 -27865.369} C_VEL
LIN {X 0,Y 89.832,Z 560.636,A -85,B 0,C 180,E1 -27873.265,E2 -27873.265} C_VEL
LIN {X 0,Y 86.469,Z 551.135,A -85,B 0,C 180,E1 -27881.027,E2 -27881.027} C_VEL
LIN {X 0,Y 84.589,Z 539.54,A -85,B 0,C 180,E1 -27889.225,E2 -27889.225} C_VEL
LIN {X 0,Y 84.052,Z 531.474,A -85,B 0,C 180,E1 -27894,E2 -27894} C_VEL
LIN {X 0,Y 83.758,Z 520.558,A -85,B 0,C 180,E1 -27899.398,E2 -27899.398} C_VEL
LIN {X 0,Y 83.818,Z 508.532,A -85,B 0,C 180,E1 -27904.207,E2 -27904.207} C_VEL
LIN {X 0,Y 84.262,Z 495.139,A -85,B 0,C 180,E1 -27908.392,E2 -27908.392} C_VEL
LIN {X 0,Y 84.718,Z 480.252,A -85,B 0,C 180,E1 -27911.817,E2 -27911.817} C_VEL
LIN {X 0,Y 85.15,Z 448.787,A -85,B 0,C 180,E1 -27917.744,E2 -27917.744} C_VEL
LIN {X 0,Y 84.455,Z 441.166,A -85,B 0,C 180,E1 -27918.991,E2 -27918.991} C_VEL
LIN {X 0,Y 82.677,Z 433.628,A -85,B 0,C 180,E1 -27920.069,E2 -27920.069} C_VEL
LIN {X 0,Y 78.146,Z 418.606,A -85,B 0,C 180,E1 -27922.165,E2 -27922.165} C_VEL
LIN {X 0,Y 73.824,Z 400.641,A -85,B 0,C 180,E1 -27925.07,E2 -27925.07} C_VEL
LIN {X 0,Y 73.224,Z 397.358,A -85,B 0,C 180,E1 -27925.773,E2 -27925.773} C_VEL
LIN {X 0,Y 72.303,Z 397.477,A -85,B 0,C 180,E1 -27938.948,E2 -27938.948} C_VEL
LIN {X 0,Y 72.253,Z 397.484,A -85,B 0,C 180,E1 -27947.079,E2 -27947.079} C_VEL
LIN {X 0,Y 72.304,Z 397.479,A -85,B 0,C 180,E1 -27954.316,E2 -27954.316} C_VEL
LIN {X 0,Y 72.378,Z 397.463,A -85,B 0,C 180,E1 -27960.947,E2 -27960.947} C_VEL
LIN {X 0,Y 72.397,Z 397.459,A -85,B 0,C 180,E1 -27967.144,E2 -27967.144} C_VEL
LIN {X 0,Y 72.723,Z 397.421,A -85,B 0,C 180,E1 -27975.104,E2 -27975.104} C_VEL
LIN {X 0,Y 72.86,Z 397.405,A -85,B 0,C 180,E1 -27978.871,E2 -27978.871} C_VEL
LIN {X 0,Y 73.573,Z 397.321,A -85,B 0,C 180,E1 -27989.994,E2 -27989.994} C_VEL
